LIN {X 0,Y 552.343,Z 361.925,A -85,B 0,C 180,E1 26679.853,E2 26679.853} C_VEL
LIN {X 0,Y 552.316,Z 361.93,A -85,B 0,C 180,E1 26676.515,E2 26676.515} C_VEL
LIN {X 0,Y 552.306,Z 361.936,A -85,B 0,C 180,E1 26673.143,E2 26673.143} C_VEL
LIN {X 0,Y 552.345,Z 361.928,A -85,B 0,C 180,E1 26669.855,E2 26669.855} C_VEL
LIN {X 0,Y 552.293,Z 361.931,A -85,B 0,C 180,E1 26666.589,E2 26666.589} C_VEL
LIN {X 0,Y 552.33,Z 361.932,A -85,B 0,C 180,E1 26663.244,E2 26663.244} C_VEL
LIN {X 0,Y 552.306,Z 361.932,A -85,B 0,C 180,E1 26660.008,E2 26660.008} C_VEL
LIN {X 0,Y 552.29,Z 361.935,A -85,B 0,C 180,E1 26656.621,E2 26656.621} C_VEL
LIN {X 0,Y 552.342,Z 361.931,A -85,B 0,C 180,E1 26653.398,E2 26653.398} C_VEL
LIN {X 0,Y 552.279,Z 361.932,A -85,B 0,C 180,E1 26650.22,E2 26650.22} C_VEL
LIN {X 0,Y 552.338,Z 361.933,A -85,B 0,C 180,E1 26646.967,E2 26646.967} C_VEL
LIN {X 0,Y 552.28,Z 361.935,A -85,B 0,C 180,E1 26643.737,E2 26643.737} C_VEL
LIN {X 0,Y 552.285,Z 361.937,A -85,B 0,C 180,E1 26640.311,E2 26640.311} C_VEL
LIN {X 0,Y 552.292,Z 361.933,A -85,B 0,C 180,E1 26637.302,E2 26637.302} C_VEL
LIN {X 0,Y 552.269,Z 361.935,A -85,B 0,C 180,E1 26633.973,E2 26633.973} C_VEL
LIN {X 0,Y 552.307,Z 361.936,A -85,B 0,C 180,E1 26630.939,E2 26630.939} C_VEL
LIN {X 0,Y 552.259,Z 361.937,A -85,B 0,C 180,E1 26627.665,E2 26627.665} C_VEL
LIN {X 0,Y 552.332,Z 361.933,A -85,B 0,C 180,E1 26624.46,E2 26624.46} C_VEL
LIN {X 0,Y 552.255,Z 361.936,A -85,B 0,C 180,E1 26621.227,E2 26621.227} C_VEL
LIN {X 0,Y 552.295,Z 361.933,A -85,B 0,C 180,E1 26617.945,E2 26617.945} C_VEL
LIN {X 0,Y 552.264,Z 361.927,A -85,B 0,C 180,E1 26614.935,E2 26614.935} C_VEL
LIN {X 0,Y 552.281,Z 361.934,A -85,B 0,C 180,E1 26611.567,E2 26611.567} C_VEL
LIN {X 0,Y 552.273,Z 361.928,A -85,B 0,C 180,E1 26608.695,E2 26608.695} C_VEL
LIN {X 0,Y 552.276,Z 361.929,A -85,B 0,C 180,E1 26605.23,E2 26605.23} C_VEL
LIN {X 0,Y 552.317,Z 361.938,A -85,B 0,C 180,E1 26602.112,E2 26602.112} C_VEL
LIN {X 0,Y 552.276,Z 361.935,A -85,B 0,C 180,E1 26598.857,E2 26598.857} C_VEL
LIN {X 0,Y 552.345,Z 361.921,A -85,B 0,C 180,E1 26595.64,E2 26595.64} C_VEL
LIN {X 0,Y 552.28,Z 361.923,A -85,B 0,C 180,E1 26592.384,E2 26592.384} C_VEL
LIN {X 0,Y 552.364,Z 362.227,A -85,B 0,C 180,E1 26591.86,E2 26591.86} C_VEL
LIN {X 0,Y 554.756,Z 368.091,A -85,B 0,C 180,E1 26591.269,E2 26591.269} C_VEL
LIN {X 0,Y 560.698,Z 379.842,A -85,B 0,C 180,E1 26590.068,E2 26590.068} C_VEL
LIN {X 0,Y 561.621,Z 381.954,A -85,B 0,C 180,E1 26589.855,E2 26589.855} C_VEL
LIN {X 0,Y 560.215,Z 433.691,A -85,B 0,C 180,E1 26586.78,E2 26586.78} C_VEL
LIN {X 0,Y 559.86,Z 455.296,A -85,B 0,C 180,E1 26585.548,E2 26585.548} C_VEL
LIN {X 0,Y 561.193,Z 465.51,A -85,B 0,C 180,E1 26585.289,E2 26585.289} C_VEL
LIN {X 0,Y 559.582,Z 691.156,A -85,B 0,C 180,E1 26581.995,E2 26581.995} C_VEL
LIN {X 0,Y 559.04,Z 762.319,A -85,B 0,C 180,E1 26580.945,E2 26580.945} C_VEL
LIN {X 0,Y 558.579,Z 783.876,A -85,B 0,C 180,E1 26580.433,E2 26580.433} C_VEL
LIN {X 0,Y 558.05,Z 805.556,A -85,B 0,C 180,E1 26579.723,E2 26579.723} C_VEL
LIN {X 0,Y 557.439,Z 826.444,A -85,B 0,C 180,E1 26578.846,E2 26578.846} C_VEL
LIN {X 0,Y 556.74,Z 845.795,A -85,B 0,C 180,E1 26577.833,E2 26577.833} C_VEL
LIN {X 0,Y 555.982,Z 866.365,A -85,B 0,C 180,E1 26576.542,E2 26576.542} C_VEL
LIN {X 0,Y 555.24,Z 885.138,A -85,B 0,C 180,E1 26575.147,E2 26575.147} C_VEL
LIN {X 0,Y 554.547,Z 902.924,A -85,B 0,C 180,E1 26573.593,E2 26573.593} C_VEL
LIN {X 0,Y 553.91,Z 919.52,A -85,B 0,C 180,E1 26571.904,E2 26571.904} C_VEL
LIN {X 0,Y 553.324,Z 935.884,A -85,B 0,C 180,E1 26569.968,E2 26569.968} C_VEL
LIN {X 0,Y 552.863,Z 950.053,A -85,B 0,C 180,E1 26568.013,E2 26568.013} C_VEL
LIN {X 0,Y 552.505,Z 962.742,A -85,B 0,C 180,E1 26565.965,E2 26565.965} C_VEL
LIN {X 0,Y 552.256,Z 973.338,A -85,B 0,C 180,E1 26563.932,E2 26563.932} C_VEL
LIN {X 0,Y 552.08,Z 983.072,A -85,B 0,C 180,E1 26561.702,E2 26561.702} C_VEL
LIN {X 0,Y 551.98,Z 990.592,A -85,B 0,C 180,E1 26559.592,E2 26559.592} C_VEL
LIN {X 0,Y 551.925,Z 996.4,A -85,B 0,C 180,E1 26557.494,E2 26557.494} C_VEL
LIN {X 0,Y 551.904,Z 1000.985,A -85,B 0,C 180,E1 26555.301,E2 26555.301} C_VEL
LIN {X 0,Y 551.907,Z 1003.785,A -85,B 0,C 180,E1 26553.22,E2 26553.22} C_VEL
LIN {X 0,Y 551.904,Z 1005.306,A -85,B 0,C 180,E1 26550.935,E2 26550.935} C_VEL
LIN {X 0,Y 551.909,Z 1005.238,A -85,B 0,C 180,E1 26548.755,E2 26548.755} C_VEL
LIN {X 0,Y 551.915,Z 1003.544,A -85,B 0,C 180,E1 26546.558,E2 26546.558} C_VEL
LIN {X 0,Y 551.924,Z 1000.222,A -85,B 0,C 180,E1 26544.283,E2 26544.283} C_VEL
LIN {X 0,Y 551.946,Z 995.639,A -85,B 0,C 180,E1 26542.193,E2 26542.193} C_VEL
LIN {X 0,Y 552.003,Z 989.18,A -85,B 0,C 180,E1 26539.987,E2 26539.987} C_VEL
LIN {X 0,Y 552.116,Z 981.437,A -85,B 0,C 180,E1 26537.875,E2 26537.875} C_VEL
LIN {X 0,Y 552.296,Z 971.783,A -85,B 0,C 180,E1 26535.748,E2 26535.748} C_VEL
LIN {X 0,Y 552.58,Z 960.206,A -85,B 0,C 180,E1 26533.606,E2 26533.606} C_VEL
LIN {X 0,Y 552.936,Z 947.891,A -85,B 0,C 180,E1 26531.663,E2 26531.663} C_VEL
LIN {X 0,Y 553.409,Z 933.339,A -85,B 0,C 180,E1 26529.705,E2 26529.705} C_VEL
LIN {X 0,Y 553.971,Z 917.685,A -85,B 0,C 180,E1 26527.897,E2 26527.897} C_VEL
LIN {X 0,Y 554.661,Z 899.915,A -85,B 0,C 180,E1 26526.131,E2 26526.131} C_VEL
LIN {X 0,Y 555.379,Z 881.773,A -85,B 0,C 180,E1 26524.588,E2 26524.588} C_VEL
LIN {X 0,Y 556.106,Z 863.135,A -85,B 0,C 180,E1 26523.235,E2 26523.235} C_VEL
LIN {X 0,Y 556.812,Z 843.818,A -85,B 0,C 180,E1 26522.055,E2 26522.055} C_VEL
LIN {X 0,Y 557.491,Z 823.944,A -85,B 0,C 180,E1 26521.041,E2 26521.041} C_VEL
LIN {X 0,Y 558.103,Z 804.103,A -85,B 0,C 180,E1 26520.222,E2 26520.222} C_VEL
LIN {X 0,Y 558.602,Z 782.228,A -85,B 0,C 180,E1 26519.521,E2 26519.521} C_VEL
LIN {X 0,Y 559.058,Z 760.348,A -85,B 0,C 180,E1 26519.022,E2 26519.022} C_VEL
LIN {X 0,Y 560.653,Z 537.271,A -85,B 0,C 180,E1 26515.768,E2 26515.768} C_VEL
LIN {X 0,Y 561.011,Z 462.845,A -85,B 0,C 180,E1 26514.657,E2 26514.657} C_VEL
LIN {X 0,Y 559.765,Z 453.839,A -85,B 0,C 180,E1 26514.392,E2 26514.392} C_VEL
LIN {X 0,Y 561.186,Z 397.807,A -85,B 0,C 180,E1 26511.099,E2 26511.099} C_VEL
LIN {X 0,Y 561.58,Z 381.583,A -85,B 0,C 180,E1 26510.118,E2 26510.118} C_VEL
LIN {X 0,Y 555.25,Z 369.007,A -85,B 0,C 180,E1 26508.825,E2 26508.825} C_VEL
LIN {X 0,Y 552.385,Z 362.34,A -85,B 0,C 180,E1 26508.161,E2 26508.161} C_VEL
LIN {X 0,Y 552.29,Z 361.923,A -85,B 0,C 180,E1 26507.811,E2 26507.811} C_VEL
LIN {X 0,Y 552.321,Z 361.927,A -85,B 0,C 180,E1 26504.654,E2 26504.654} C_VEL
LIN {X 0,Y 552.276,Z 361.935,A -85,B 0,C 180,E1 26501.361,E2 26501.361} C_VEL
LIN {X 0,Y 552.342,Z 361.936,A -85,B 0,C 180,E1 26498.118,E2 26498.118} C_VEL
LIN {X 0,Y 552.271,Z 361.93,A -85,B 0,C 180,E1 26494.897,E2 26494.897} C_VEL
LIN {X 0,Y 552.308,Z 361.928,A -85,B 0,C 180,E1 26491.668,E2 26491.668} C_VEL
LIN {X 0,Y 552.268,Z 361.934,A -85,B 0,C 180,E1 26488.67,E2 26488.67} C_VEL
LIN {X 0,Y 552.283,Z 361.926,A -85,B 0,C 180,E1 26485.293,E2 26485.293} C_VEL
LIN {X 0,Y 552.279,Z 361.932,A -85,B 0,C 180,E1 26482.233,E2 26482.233} C_VEL
LIN {X 0,Y 552.263,Z 361.936,A -85,B 0,C 180,E1 26478.909,E2 26478.909} C_VEL
LIN {X 0,Y 552.291,Z 361.939,A -85,B 0,C 180,E1 26475.864,E2 26475.864} C_VEL
LIN {X 0,Y 552.259,Z 361.938,A -85,B 0,C 180,E1 26472.644,E2 26472.644} C_VEL
LIN {X 0,Y 552.322,Z 361.937,A -85,B 0,C 180,E1 26469.482,E2 26469.482} C_VEL
LIN {X 0,Y 552.261,Z 361.935,A -85,B 0,C 180,E1 26466.34,E2 26466.34} C_VEL
LIN {X 0,Y 552.332,Z 361.932,A -85,B 0,C 180,E1 26463.113,E2 26463.113} C_VEL
LIN {X 0,Y 552.266,Z 361.937,A -85,B 0,C 180,E1 26460,E2 26460} C_VEL
LIN {X 0,Y 552.317,Z 361.935,A -85,B 0,C 180,E1 26456.723,E2 26456.723} C_VEL
LIN {X 0,Y 552.281,Z 361.931,A -85,B 0,C 180,E1 26453.555,E2 26453.555} C_VEL
LIN {X 0,Y 552.283,Z 361.931,A -85,B 0,C 180,E1 26450.096,E2 26450.096} C_VEL
LIN {X 0,Y 552.331,Z 361.938,A -85,B 0,C 180,E1 26446.922,E2 26446.922} C_VEL
LIN {X 0,Y 552.281,Z 361.935,A -85,B 0,C 180,E1 26443.703,E2 26443.703} C_VEL
LIN {X 0,Y 552.342,Z 361.933,A -85,B 0,C 180,E1 26440.434,E2 26440.434} C_VEL
LIN {X 0,Y 552.29,Z 361.934,A -85,B 0,C 180,E1 26437.206,E2 26437.206} C_VEL
LIN {X 0,Y 552.307,Z 361.93,A -85,B 0,C 180,E1 26433.786,E2 26433.786} C_VEL
LIN {X 0,Y 552.325,Z 361.933,A -85,B 0,C 180,E1 26432.641,E2 26432.641} C_VEL
LIN {X 0,Y 551.377,Z 362.054,A -85,B 0,C 180,E1 26431.841,E2 26431.841} C_VEL
LIN {X 0,Y 544.88,Z 362.854,A -85,B 0,C 180,E1 26429.597,E2 26429.597} C_VEL
LIN {X 0,Y 544.354,Z 362.92,A -85,B 0,C 180,E1 26429.012,E2 26429.012} C_VEL
LIN {X 0,Y 544.385,Z 362.919,A -85,B 0,C 180,E1 26425.677,E2 26425.677} C_VEL
LIN {X 0,Y 544.393,Z 362.912,A -85,B 0,C 180,E1 26422.327,E2 26422.327} C_VEL
LIN {X 0,Y 544.361,Z 362.922,A -85,B 0,C 180,E1 26419.01,E2 26419.01} C_VEL
LIN {X 0,Y 544.404,Z 362.907,A -85,B 0,C 180,E1 26415.74,E2 26415.74} C_VEL
LIN {X 0,Y 544.371,Z 362.925,A -85,B 0,C 180,E1 26412.408,E2 26412.408} C_VEL
LIN {X 0,Y 544.373,Z 362.924,A -85,B 0,C 180,E1 26408.909,E2 26408.909} C_VEL
LIN {X 0,Y 544.402,Z 362.924,A -85,B 0,C 180,E1 26405.548,E2 26405.548} C_VEL
LIN {X 0,Y 544.431,Z 363.119,A -85,B 0,C 180,E1 26403.177,E2 26403.177} C_VEL
LIN {X 0,Y 548.647,Z 375.762,A -85,B 0,C 180,E1 26401.572,E2 26401.572} C_VEL
LIN {X 0,Y 549.438,Z 378.934,A -85,B 0,C 180,E1 26401.237,E2 26401.237} C_VEL
LIN {X 0,Y 549.463,Z 383.628,A -85,B 0,C 180,E1 26400.87,E2 26400.87} C_VEL
LIN {X 0,Y 551.825,Z 395.845,A -85,B 0,C 180,E1 26400.533,E2 26400.533} C_VEL
LIN {X 0,Y 550.089,Z 643.165,A -85,B 0,C 180,E1 26397,E2 26397} C_VEL
LIN {X 0,Y 549.682,Z 663.581,A -85,B 0,C 180,E1 26396.524,E2 26396.524} C_VEL
LIN {X 0,Y 549.19,Z 683.218,A -85,B 0,C 180,E1 26395.877,E2 26395.877} C_VEL
LIN {X 0,Y 548.592,Z 703.287,A -85,B 0,C 180,E1 26395.011,E2 26395.011} C_VEL
LIN {X 0,Y 547.936,Z 721.879,A -85,B 0,C 180,E1 26394.009,E2 26394.009} C_VEL
LIN {X 0,Y 547.252,Z 740.465,A -85,B 0,C 180,E1 26392.786,E2 26392.786} C_VEL
LIN {X 0,Y 546.545,Z 758.589,A -85,B 0,C 180,E1 26391.347,E2 26391.347} C_VEL
LIN {X 0,Y 545.911,Z 774.895,A -85,B 0,C 180,E1 26389.803,E2 26389.803} C_VEL
LIN {X 0,Y 545.352,Z 789.659,A -85,B 0,C 180,E1 26388.158,E2 26388.158} C_VEL
LIN {X 0,Y 544.9,Z 803.014,A -85,B 0,C 180,E1 26386.412,E2 26386.412} C_VEL
LIN {X 0,Y 544.518,Z 815.631,A -85,B 0,C 180,E1 26384.459,E2 26384.459} C_VEL
LIN {X 0,Y 544.256,Z 826.628,A -85,B 0,C 180,E1 26382.41,E2 26382.41} C_VEL
LIN {X 0,Y 544.081,Z 835.589,A -85,B 0,C 180,E1 26380.374,E2 26380.374} C_VEL
LIN {X 0,Y 543.986,Z 843.067,A -85,B 0,C 180,E1 26378.241,E2 26378.241} C_VEL
LIN {X 0,Y 543.936,Z 848.903,A -85,B 0,C 180,E1 26376.013,E2 26376.013} C_VEL
LIN {X 0,Y 543.918,Z 852.677,A -85,B 0,C 180,E1 26373.899,E2 26373.899} C_VEL
LIN {X 0,Y 543.91,Z 854.847,A -85,B 0,C 180,E1 26371.79,E2 26371.79} C_VEL
LIN {X 0,Y 543.904,Z 855.449,A -85,B 0,C 180,E1 26369.684,E2 26369.684} C_VEL
LIN {X 0,Y 543.905,Z 854.492,A -85,B 0,C 180,E1 26367.577,E2 26367.577} C_VEL
LIN {X 0,Y 543.918,Z 851.699,A -85,B 0,C 180,E1 26365.361,E2 26365.361} C_VEL
LIN {X 0,Y 543.945,Z 847.346,A -85,B 0,C 180,E1 26363.244,E2 26363.244} C_VEL
LIN {X 0,Y 543.998,Z 841.271,A -85,B 0,C 180,E1 26361.119,E2 26361.119} C_VEL
LIN {X 0,Y 544.105,Z 833.793,A -85,B 0,C 180,E1 26359.09,E2 26359.09} C_VEL
LIN {X 0,Y 544.307,Z 824.452,A -85,B 0,C 180,E1 26357.051,E2 26357.051} C_VEL
LIN {X 0,Y 544.578,Z 813.591,A -85,B 0,C 180,E1 26355.106,E2 26355.106} C_VEL
LIN {X 0,Y 544.949,Z 801.32,A -85,B 0,C 180,E1 26353.26,E2 26353.26} C_VEL
LIN {X 0,Y 545.419,Z 787.628,A -85,B 0,C 180,E1 26351.511,E2 26351.511} C_VEL
LIN {X 0,Y 546.016,Z 771.787,A -85,B 0,C 180,E1 26349.796,E2 26349.796} C_VEL
LIN {X 0,Y 546.675,Z 755.081,A -85,B 0,C 180,E1 26348.269,E2 26348.269} C_VEL
LIN {X 0,Y 547.359,Z 737.607,A -85,B 0,C 180,E1 26346.925,E2 26346.925} C_VEL
LIN {X 0,Y 548.021,Z 719.612,A -85,B 0,C 180,E1 26345.765,E2 26345.765} C_VEL
LIN {X 0,Y 548.681,Z 700.505,A -85,B 0,C 180,E1 26344.762,E2 26344.762} C_VEL
LIN {X 0,Y 549.259,Z 681.058,A -85,B 0,C 180,E1 26343.952,E2 26343.952} C_VEL
LIN {X 0,Y 549.733,Z 660.673,A -85,B 0,C 180,E1 26343.307,E2 26343.307} C_VEL
LIN {X 0,Y 550.118,Z 639.409,A -85,B 0,C 180,E1 26342.848,E2 26342.848} C_VEL
LIN {X 0,Y 551.822,Z 394.728,A -85,B 0,C 180,E1 26339.361,E2 26339.361} C_VEL
LIN {X 0,Y 549.369,Z 382.831,A -85,B 0,C 180,E1 26339.001,E2 26339.001} C_VEL
LIN {X 0,Y 549.407,Z 378.116,A -85,B 0,C 180,E1 26338.598,E2 26338.598} C_VEL
LIN {X 0,Y 544.904,Z 364.895,A -85,B 0,C 180,E1 26336.989,E2 26336.989} C_VEL
LIN {X 0,Y 544.412,Z 363.01,A -85,B 0,C 180,E1 26336.695,E2 26336.695} C_VEL
LIN {X 0,Y 544.373,Z 362.914,A -85,B 0,C 180,E1 26333.353,E2 26333.353} C_VEL
LIN {X 0,Y 544.403,Z 362.917,A -85,B 0,C 180,E1 26329.985,E2 26329.985} C_VEL
LIN {X 0,Y 544.403,Z 362.92,A -85,B 0,C 180,E1 26326.508,E2 26326.508} C_VEL
LIN {X 0,Y 544.366,Z 362.921,A -85,B 0,C 180,E1 26323.187,E2 26323.187} C_VEL
LIN {X 0,Y 544.404,Z 362.912,A -85,B 0,C 180,E1 26319.858,E2 26319.858} C_VEL
LIN {X 0,Y 544.376,Z 362.919,A -85,B 0,C 180,E1 26316.519,E2 26316.519} C_VEL
LIN {X 0,Y 544.363,Z 362.925,A -85,B 0,C 180,E1 26313.06,E2 26313.06} C_VEL
LIN {X 0,Y 544.406,Z 362.918,A -85,B 0,C 180,E1 26309.728,E2 26309.728} C_VEL
LIN {X 0,Y 544.356,Z 362.92,A -85,B 0,C 180,E1 26306.509,E2 26306.509} C_VEL
LIN {X 0,Y 544.381,Z 362.922,A -85,B 0,C 180,E1 26303.145,E2 26303.145} C_VEL
LIN {X 0,Y 544.379,Z 362.92,A -85,B 0,C 180,E1 26299.864,E2 26299.864} C_VEL
LIN {X 0,Y 544.348,Z 362.924,A -85,B 0,C 180,E1 26296.52,E2 26296.52} C_VEL
LIN {X 0,Y 544.407,Z 362.921,A -85,B 0,C 180,E1 26293.268,E2 26293.268} C_VEL
LIN {X 0,Y 544.342,Z 362.92,A -85,B 0,C 180,E1 26290.05,E2 26290.05} C_VEL
LIN {X 0,Y 544.375,Z 362.92,A -85,B 0,C 180,E1 26286.751,E2 26286.751} C_VEL
LIN {X 0,Y 544.35,Z 362.924,A -85,B 0,C 180,E1 26283.581,E2 26283.581} C_VEL
LIN {X 0,Y 544.338,Z 362.926,A -85,B 0,C 180,E1 26280.211,E2 26280.211} C_VEL
LIN {X 0,Y 544.379,Z 362.921,A -85,B 0,C 180,E1 26277.052,E2 26277.052} C_VEL
LIN {X 0,Y 544.325,Z 362.924,A -85,B 0,C 180,E1 26273.779,E2 26273.779} C_VEL
LIN {X 0,Y 544.394,Z 362.926,A -85,B 0,C 180,E1 26270.592,E2 26270.592} C_VEL
LIN {X 0,Y 544.322,Z 362.926,A -85,B 0,C 180,E1 26267.374,E2 26267.374} C_VEL
LIN {X 0,Y 544.344,Z 362.928,A -85,B 0,C 180,E1 26264.007,E2 26264.007} C_VEL
LIN {X 0,Y 544.333,Z 362.924,A -85,B 0,C 180,E1 26260.916,E2 26260.916} C_VEL
LIN {X 0,Y 544.323,Z 362.921,A -85,B 0,C 180,E1 26257.498,E2 26257.498} C_VEL
LIN {X 0,Y 544.385,Z 362.915,A -85,B 0,C 180,E1 26254.313,E2 26254.313} C_VEL
LIN {X 0,Y 544.324,Z 362.924,A -85,B 0,C 180,E1 26251.112,E2 26251.112} C_VEL
LIN {X 0,Y 544.399,Z 362.92,A -85,B 0,C 180,E1 26247.942,E2 26247.942} C_VEL
LIN {X 0,Y 544.332,Z 362.918,A -85,B 0,C 180,E1 26244.776,E2 26244.776} C_VEL
LIN {X 0,Y 544.372,Z 362.922,A -85,B 0,C 180,E1 26241.478,E2 26241.478} C_VEL
LIN {X 0,Y 544.351,Z 362.925,A -85,B 0,C 180,E1 26238.324,E2 26238.324} C_VEL
LIN {X 0,Y 544.351,Z 362.922,A -85,B 0,C 180,E1 26234.996,E2 26234.996} C_VEL
LIN {X 0,Y 544.375,Z 363.16,A -85,B 0,C 180,E1 26232.45,E2 26232.45} C_VEL
LIN {X 0,Y 545.681,Z 366.42,A -85,B 0,C 180,E1 26232.091,E2 26232.091} C_VEL
LIN {X 0,Y 555.056,Z 385.798,A -85,B 0,C 180,E1 26230.175,E2 26230.175} C_VEL
LIN {X 0,Y 553.444,Z 437.914,A -85,B 0,C 180,E1 26227.046,E2 26227.046} C_VEL
LIN {X 0,Y 553.129,Z 455.298,A -85,B 0,C 180,E1 26226.048,E2 26226.048} C_VEL
LIN {X 0,Y 554.65,Z 466.908,A -85,B 0,C 180,E1 26225.747,E2 26225.747} C_VEL
LIN {X 0,Y 552.786,Z 692.683,A -85,B 0,C 180,E1 26222.413,E2 26222.413} C_VEL
LIN {X 0,Y 552.171,Z 762.512,A -85,B 0,C 180,E1 26221.369,E2 26221.369} C_VEL
LIN {X 0,Y 551.64,Z 784.137,A -85,B 0,C 180,E1 26220.849,E2 26220.849} C_VEL
LIN {X 0,Y 551.017,Z 806.292,A -85,B 0,C 180,E1 26220.111,E2 26220.111} C_VEL
LIN {X 0,Y 550.331,Z 826.443,A -85,B 0,C 180,E1 26219.254,E2 26219.254} C_VEL
LIN {X 0,Y 549.538,Z 845.798,A -85,B 0,C 180,E1 26218.23,E2 26218.23} C_VEL
LIN {X 0,Y 548.656,Z 866.361,A -85,B 0,C 180,E1 26216.925,E2 26216.925} C_VEL
LIN {X 0,Y 547.804,Z 885.135,A -85,B 0,C 180,E1 26215.513,E2 26215.513} C_VEL
LIN {X 0,Y 547.003,Z 902.926,A -85,B 0,C 180,E1 26213.939,E2 26213.939} C_VEL
LIN {X 0,Y 546.265,Z 919.196,A -85,B 0,C 180,E1 26212.263,E2 26212.263} C_VEL
LIN {X 0,Y 545.603,Z 935.035,A -85,B 0,C 180,E1 26210.375,E2 26210.375} C_VEL
LIN {X 0,Y 545.096,Z 948.639,A -85,B 0,C 180,E1 26208.5,E2 26208.5} C_VEL
LIN {X 0,Y 544.662,Z 961.471,A -85,B 0,C 180,E1 26206.42,E2 26206.42} C_VEL
LIN {X 0,Y 544.34,Z 972.82,A -85,B 0,C 180,E1 26204.248,E2 26204.248} C_VEL
LIN {X 0,Y 544.135,Z 982.257,A -85,B 0,C 180,E1 26202.091,E2 26202.091} C_VEL
LIN {X 0,Y 544.009,Z 989.886,A -85,B 0,C 180,E1 26199.948,E2 26199.948} C_VEL
LIN {X 0,Y 543.942,Z 996.146,A -85,B 0,C 180,E1 26197.711,E2 26197.711} C_VEL
LIN {X 0,Y 543.915,Z 1000.824,A -85,B 0,C 180,E1 26195.485,E2 26195.485} C_VEL
LIN {X 0,Y 543.91,Z 1003.785,A -85,B 0,C 180,E1 26193.267,E2 26193.267} C_VEL
LIN {X 0,Y 543.905,Z 1005.306,A -85,B 0,C 180,E1 26190.948,E2 26190.948} C_VEL
LIN {X 0,Y 543.908,Z 1005.238,A -85,B 0,C 180,E1 26188.736,E2 26188.736} C_VEL
LIN {X 0,Y 543.913,Z 1003.56,A -85,B 0,C 180,E1 26186.523,E2 26186.523} C_VEL
LIN {X 0,Y 543.927,Z 1000.222,A -85,B 0,C 180,E1 26184.198,E2 26184.198} C_VEL
LIN {X 0,Y 543.958,Z 995.639,A -85,B 0,C 180,E1 26182.077,E2 26182.077} C_VEL
LIN {X 0,Y 544.03,Z 989.181,A -85,B 0,C 180,E1 26179.839,E2 26179.839} C_VEL
LIN {X 0,Y 544.161,Z 981.436,A -85,B 0,C 180,E1 26177.695,E2 26177.695} C_VEL
LIN {X 0,Y 544.377,Z 971.784,A -85,B 0,C 180,E1 26175.537,E2 26175.537} C_VEL
LIN {X 0,Y 544.706,Z 960.206,A -85,B 0,C 180,E1 26173.362,E2 26173.362} C_VEL
LIN {X 0,Y 545.123,Z 947.889,A -85,B 0,C 180,E1 26171.391,E2 26171.391} C_VEL
LIN {X 0,Y 545.673,Z 933.34,A -85,B 0,C 180,E1 26169.405,E2 26169.405} C_VEL
LIN {X 0,Y 546.304,Z 918.191,A -85,B 0,C 180,E1 26167.627,E2 26167.627} C_VEL
LIN {X 0,Y 547.107,Z 900.519,A -85,B 0,C 180,E1 26165.838,E2 26165.838} C_VEL
LIN {X 0,Y 547.914,Z 883.071,A -85,B 0,C 180,E1 26164.32,E2 26164.32} C_VEL
LIN {X 0,Y 548.728,Z 864.64,A -85,B 0,C 180,E1 26162.954,E2 26162.954} C_VEL
LIN {X 0,Y 549.583,Z 844.709,A -85,B 0,C 180,E1 26161.707,E2 26161.707} C_VEL
LIN {X 0,Y 550.38,Z 824.652,A -85,B 0,C 180,E1 26160.663,E2 26160.663} C_VEL
LIN {X 0,Y 551.074,Z 804.84,A -85,B 0,C 180,E1 26159.833,E2 26159.833} C_VEL
LIN {X 0,Y 551.669,Z 782.618,A -85,B 0,C 180,E1 26159.108,E2 26159.108} C_VEL
LIN {X 0,Y 552.189,Z 760.883,A -85,B 0,C 180,E1 26158.602,E2 26158.602} C_VEL
LIN {X 0,Y 554.023,Z 539.306,A -85,B 0,C 180,E1 26155.332,E2 26155.332} C_VEL
LIN {X 0,Y 554.48,Z 464.261,A -85,B 0,C 180,E1 26154.199,E2 26154.199} C_VEL
LIN {X 0,Y 553.035,Z 453.865,A -85,B 0,C 180,E1 26153.891,E2 26153.891} C_VEL
LIN {X 0,Y 554.652,Z 398.862,A -85,B 0,C 180,E1 26150.619,E2 26150.619} C_VEL
LIN {X 0,Y 555.03,Z 385.441,A -85,B 0,C 180,E1 26149.801,E2 26149.801} C_VEL
LIN {X 0,Y 546.189,Z 367.32,A -85,B 0,C 180,E1 26148.007,E2 26148.007} C_VEL
LIN {X 0,Y 544.414,Z 363.375,A -85,B 0,C 180,E1 26147.587,E2 26147.587} C_VEL
LIN {X 0,Y 544.341,Z 362.909,A -85,B 0,C 180,E1 26147.284,E2 26147.284} C_VEL
LIN {X 0,Y 544.37,Z 362.912,A -85,B 0,C 180,E1 26143.952,E2 26143.952} C_VEL
LIN {X 0,Y 544.351,Z 362.919,A -85,B 0,C 180,E1 26140.828,E2 26140.828} C_VEL
LIN {X 0,Y 544.341,Z 362.926,A -85,B 0,C 180,E1 26137.444,E2 26137.444} C_VEL
LIN {X 0,Y 544.391,Z 362.917,A -85,B 0,C 180,E1 26134.195,E2 26134.195} C_VEL
LIN {X 0,Y 544.326,Z 362.915,A -85,B 0,C 180,E1 26130.938,E2 26130.938} C_VEL
LIN {X 0,Y 544.383,Z 362.928,A -85,B 0,C 180,E1 26127.689,E2 26127.689} C_VEL
LIN {X 0,Y 544.325,Z 362.913,A -85,B 0,C 180,E1 26124.528,E2 26124.528} C_VEL
LIN {X 0,Y 544.334,Z 362.928,A -85,B 0,C 180,E1 26121.09,E2 26121.09} C_VEL
LIN {X 0,Y 544.35,Z 362.924,A -85,B 0,C 180,E1 26117.973,E2 26117.973} C_VEL
LIN {X 0,Y 544.317,Z 362.926,A -85,B 0,C 180,E1 26114.684,E2 26114.684} C_VEL
LIN {X 0,Y 544.389,Z 362.921,A -85,B 0,C 180,E1 26111.441,E2 26111.441} C_VEL
LIN {X 0,Y 544.319,Z 362.926,A -85,B 0,C 180,E1 26108.237,E2 26108.237} C_VEL
LIN {X 0,Y 544.383,Z 362.925,A -85,B 0,C 180,E1 26105.058,E2 26105.058} C_VEL
LIN {X 0,Y 544.331,Z 362.923,A -85,B 0,C 180,E1 26101.894,E2 26101.894} C_VEL
LIN {X 0,Y 544.35,Z 362.919,A -85,B 0,C 180,E1 26098.526,E2 26098.526} C_VEL
LIN {X 0,Y 544.36,Z 362.926,A -85,B 0,C 180,E1 26095.364,E2 26095.364} C_VEL
LIN {X 0,Y 544.339,Z 362.924,A -85,B 0,C 180,E1 26092.081,E2 26092.081} C_VEL
LIN {X 0,Y 544.398,Z 362.92,A -85,B 0,C 180,E1 26088.881,E2 26088.881} C_VEL
LIN {X 0,Y 544.338,Z 362.922,A -85,B 0,C 180,E1 26085.642,E2 26085.642} C_VEL
LIN {X 0,Y 544.395,Z 362.92,A -85,B 0,C 180,E1 26082.359,E2 26082.359} C_VEL
LIN {X 0,Y 544.355,Z 362.925,A -85,B 0,C 180,E1 26079.125,E2 26079.125} C_VEL
LIN {X 0,Y 544.352,Z 362.922,A -85,B 0,C 180,E1 26075.637,E2 26075.637} C_VEL
LIN {X 0,Y 544.405,Z 362.921,A -85,B 0,C 180,E1 26072.43,E2 26072.43} C_VEL
LIN {X 0,Y 544.353,Z 362.919,A -85,B 0,C 180,E1 26069.172,E2 26069.172} C_VEL
LIN {X 0,Y 544.354,Z 362.92,A -85,B 0,C 180,E1 26069.012,E2 26069.012} C_VEL
LIN {X 0,Y 543.393,Z 363.05,A -85,B 0,C 180,E1 26068.202,E2 26068.202} C_VEL
LIN {X 0,Y 536.877,Z 363.856,A -85,B 0,C 180,E1 26065.865,E2 26065.865} C_VEL
LIN {X 0,Y 536.422,Z 363.91,A -85,B 0,C 180,E1 26065.331,E2 26065.331} C_VEL
LIN {X 0,Y 536.465,Z 363.892,A -85,B 0,C 180,E1 26062.027,E2 26062.027} C_VEL
LIN {X 0,Y 536.426,Z 363.913,A -85,B 0,C 180,E1 26058.684,E2 26058.684} C_VEL
LIN {X 0,Y 536.437,Z 363.9,A -85,B 0,C 180,E1 26055.207,E2 26055.207} C_VEL
LIN {X 0,Y 536.462,Z 363.897,A -85,B 0,C 180,E1 26051.849,E2 26051.849} C_VEL
LIN {X 0,Y 536.429,Z 363.915,A -85,B 0,C 180,E1 26048.478,E2 26048.478} C_VEL
LIN {X 0,Y 536.453,Z 363.909,A -85,B 0,C 180,E1 26045.029,E2 26045.029} C_VEL
LIN {X 0,Y 536.497,Z 364.158,A -85,B 0,C 180,E1 26043.732,E2 26043.732} C_VEL
LIN {X 0,Y 541.522,Z 378.665,A -85,B 0,C 180,E1 26041.86,E2 26041.86} C_VEL
LIN {X 0,Y 542.341,Z 381.653,A -85,B 0,C 180,E1 26041.507,E2 26041.507} C_VEL
LIN {X 0,Y 542.494,Z 384.417,A -85,B 0,C 180,E1 26041.32,E2 26041.32} C_VEL
LIN {X 0,Y 544.927,Z 397.237,A -85,B 0,C 180,E1 26040.941,E2 26040.941} C_VEL
LIN {X 0,Y 542.962,Z 642.994,A -85,B 0,C 180,E1 26037.387,E2 26037.387} C_VEL
LIN {X 0,Y 542.502,Z 663.463,A -85,B 0,C 180,E1 26036.907,E2 26036.907} C_VEL
LIN {X 0,Y 541.952,Z 683.236,A -85,B 0,C 180,E1 26036.249,E2 26036.249} C_VEL
LIN {X 0,Y 541.268,Z 703.299,A -85,B 0,C 180,E1 26035.373,E2 26035.373} C_VEL
LIN {X 0,Y 540.524,Z 721.888,A -85,B 0,C 180,E1 26034.359,E2 26034.359} C_VEL
LIN {X 0,Y 539.754,Z 740.473,A -85,B 0,C 180,E1 26033.121,E2 26033.121} C_VEL
LIN {X 0,Y 538.948,Z 758.6,A -85,B 0,C 180,E1 26031.663,E2 26031.663} C_VEL
LIN {X 0,Y 538.22,Z 774.903,A -85,B 0,C 180,E1 26030.099,E2 26030.099} C_VEL
LIN {X 0,Y 537.577,Z 789.664,A -85,B 0,C 180,E1 26028.43,E2 26028.43} C_VEL
LIN {X 0,Y 537.057,Z 803.018,A -85,B 0,C 180,E1 26026.659,E2 26026.659} C_VEL
LIN {X 0,Y 536.617,Z 815.633,A -85,B 0,C 180,E1 26024.677,E2 26024.677} C_VEL
LIN {X 0,Y 536.313,Z 826.632,A -85,B 0,C 180,E1 26022.597,E2 26022.597} C_VEL
LIN {X 0,Y 536.113,Z 835.593,A -85,B 0,C 180,E1 26020.53,E2 26020.53} C_VEL
LIN {X 0,Y 536,Z 843.069,A -85,B 0,C 180,E1 26018.365,E2 26018.365} C_VEL
LIN {X 0,Y 535.94,Z 848.905,A -85,B 0,C 180,E1 26016.103,E2 26016.103} C_VEL
LIN {X 0,Y 535.919,Z 852.678,A -85,B 0,C 180,E1 26013.958,E2 26013.958} C_VEL
LIN {X 0,Y 535.911,Z 854.847,A -85,B 0,C 180,E1 26011.817,E2 26011.817} C_VEL
LIN {X 0,Y 535.904,Z 855.449,A -85,B 0,C 180,E1 26009.679,E2 26009.679} C_VEL
LIN {X 0,Y 535.905,Z 854.491,A -85,B 0,C 180,E1 26007.54,E2 26007.54} C_VEL
LIN {X 0,Y 535.919,Z 851.857,A -85,B 0,C 180,E1 26005.399,E2 26005.399} C_VEL
LIN {X 0,Y 535.948,Z 847.599,A -85,B 0,C 180,E1 26003.251,E2 26003.251} C_VEL
LIN {X 0,Y 536.009,Z 841.623,A -85,B 0,C 180,E1 26001.094,E2 26001.094} C_VEL
LIN {X 0,Y 536.132,Z 834.248,A -85,B 0,C 180,E1 25999.035,E2 25999.035} C_VEL
LIN {X 0,Y 536.356,Z 824.977,A -85,B 0,C 180,E1 25996.965,E2 25996.965} C_VEL
LIN {X 0,Y 536.665,Z 814.228,A -85,B 0,C 180,E1 25994.992,E2 25994.992} C_VEL
LIN {X 0,Y 537.087,Z 802.055,A -85,B 0,C 180,E1 25993.114,E2 25993.114} C_VEL
LIN {X 0,Y 537.619,Z 788.549,A -85,B 0,C 180,E1 25991.346,E2 25991.346} C_VEL
LIN {X 0,Y 538.269,Z 773.57,A -85,B 0,C 180,E1 25989.676,E2 25989.676} C_VEL
LIN {X 0,Y 538.986,Z 757.656,A -85,B 0,C 180,E1 25988.166,E2 25988.166} C_VEL
LIN {X 0,Y 539.782,Z 739.877,A -85,B 0,C 180,E1 25986.746,E2 25986.746} C_VEL
LIN {X 0,Y 540.552,Z 721.268,A -85,B 0,C 180,E1 25985.513,E2 25985.513} C_VEL
LIN {X 0,Y 541.283,Z 702.754,A -85,B 0,C 180,E1 25984.51,E2 25984.51} C_VEL
LIN {X 0,Y 541.933,Z 683.811,A -85,B 0,C 180,E1 25983.683,E2 25983.683} C_VEL
LIN {X 0,Y 542.499,Z 663.774,A -85,B 0,C 180,E1 25983.011,E2 25983.011} C_VEL
LIN {X 0,Y 542.961,Z 643.267,A -85,B 0,C 180,E1 25982.527,E2 25982.527} C_VEL
LIN {X 0,Y 544.914,Z 398.88,A -85,B 0,C 180,E1 25978.993,E2 25978.993} C_VEL
LIN {X 0,Y 544.609,Z 394.681,A -85,B 0,C 180,E1 25978.909,E2 25978.909} C_VEL
LIN {X 0,Y 542.322,Z 383.07,A -85,B 0,C 180,E1 25978.522,E2 25978.522} C_VEL
LIN {X 0,Y 542.049,Z 380.311,A -85,B 0,C 180,E1 25978.251,E2 25978.251} C_VEL
LIN {X 0,Y 537.617,Z 367.183,A -85,B 0,C 180,E1 25976.602,E2 25976.602} C_VEL
LIN {X 0,Y 536.482,Z 364.044,A -85,B 0,C 180,E1 25976.137,E2 25976.137} C_VEL
LIN {X 0,Y 536.459,Z 363.894,A -85,B 0,C 180,E1 25972.722,E2 25972.722} C_VEL
LIN {X 0,Y 536.43,Z 363.899,A -85,B 0,C 180,E1 25969.342,E2 25969.342} C_VEL
LIN {X 0,Y 536.462,Z 363.911,A -85,B 0,C 180,E1 25965.962,E2 25965.962} C_VEL
LIN {X 0,Y 536.45,Z 363.906,A -85,B 0,C 180,E1 25962.577,E2 25962.577} C_VEL
LIN {X 0,Y 536.424,Z 363.893,A -85,B 0,C 180,E1 25959.166,E2 25959.166} C_VEL
LIN {X 0,Y 536.466,Z 363.912,A -85,B 0,C 180,E1 25955.819,E2 25955.819} C_VEL
LIN {X 0,Y 536.431,Z 363.911,A -85,B 0,C 180,E1 25952.467,E2 25952.467} C_VEL
LIN {X 0,Y 536.424,Z 363.914,A -85,B 0,C 180,E1 25948.988,E2 25948.988} C_VEL
LIN {X 0,Y 536.464,Z 363.907,A -85,B 0,C 180,E1 25945.739,E2 25945.739} C_VEL
LIN {X 0,Y 536.412,Z 363.909,A -85,B 0,C 180,E1 25942.415,E2 25942.415} C_VEL
LIN {X 0,Y 536.439,Z 363.91,A -85,B 0,C 180,E1 25939.037,E2 25939.037} C_VEL
LIN {X 0,Y 536.434,Z 363.91,A -85,B 0,C 180,E1 25935.791,E2 25935.791} C_VEL
LIN {X 0,Y 536.406,Z 363.914,A -85,B 0,C 180,E1 25932.408,E2 25932.408} C_VEL
LIN {X 0,Y 536.465,Z 363.91,A -85,B 0,C 180,E1 25929.116,E2 25929.116} C_VEL
LIN {X 0,Y 536.4,Z 363.907,A -85,B 0,C 180,E1 25925.885,E2 25925.885} C_VEL
LIN {X 0,Y 536.415,Z 363.909,A -85,B 0,C 180,E1 25922.457,E2 25922.457} C_VEL
LIN {X 0,Y 536.416,Z 363.914,A -85,B 0,C 180,E1 25919.359,E2 25919.359} C_VEL
LIN {X 0,Y 536.394,Z 363.915,A -85,B 0,C 180,E1 25916.045,E2 25916.045} C_VEL
LIN {X 0,Y 536.451,Z 363.909,A -85,B 0,C 180,E1 25912.827,E2 25912.827} C_VEL
LIN {X 0,Y 536.382,Z 363.914,A -85,B 0,C 180,E1 25909.583,E2 25909.583} C_VEL
LIN {X 0,Y 536.432,Z 363.914,A -85,B 0,C 180,E1 25906.307,E2 25906.307} C_VEL
LIN {X 0,Y 536.38,Z 363.917,A -85,B 0,C 180,E1 25903.206,E2 25903.206} C_VEL
LIN {X 0,Y 536.399,Z 363.917,A -85,B 0,C 180,E1 25899.828,E2 25899.828} C_VEL
LIN {X 0,Y 536.4,Z 363.907,A -85,B 0,C 180,E1 25896.762,E2 25896.762} C_VEL
LIN {X 0,Y 536.39,Z 363.917,A -85,B 0,C 180,E1 25893.425,E2 25893.425} C_VEL
LIN {X 0,Y 536.439,Z 363.9,A -85,B 0,C 180,E1 25890.278,E2 25890.278} C_VEL
LIN {X 0,Y 536.39,Z 363.917,A -85,B 0,C 180,E1 25887.008,E2 25887.008} C_VEL
LIN {X 0,Y 536.452,Z 363.899,A -85,B 0,C 180,E1 25883.784,E2 25883.784} C_VEL
LIN {X 0,Y 536.396,Z 363.912,A -85,B 0,C 180,E1 25880.669,E2 25880.669} C_VEL
LIN {X 0,Y 536.44,Z 363.911,A -85,B 0,C 180,E1 25877.406,E2 25877.406} C_VEL
LIN {X 0,Y 536.417,Z 363.92,A -85,B 0,C 180,E1 25874.191,E2 25874.191} C_VEL
LIN {X 0,Y 536.449,Z 364.118,A -85,B 0,C 180,E1 25873.061,E2 25873.061} C_VEL
LIN {X 0,Y 537.174,Z 366.462,A -85,B 0,C 180,E1 25872.791,E2 25872.791} C_VEL
LIN {X 0,Y 548.249,Z 389.216,A -85,B 0,C 180,E1 25870.48,E2 25870.48} C_VEL
LIN {X 0,Y 547.221,Z 426.299,A -85,B 0,C 180,E1 25868.269,E2 25868.269} C_VEL
LIN {X 0,Y 546.421,Z 455.21,A -85,B 0,C 180,E1 25866.565,E2 25866.565} C_VEL
LIN {X 0,Y 548.144,Z 468.258,A -85,B 0,C 180,E1 25866.216,E2 25866.216} C_VEL
LIN {X 0,Y 546.023,Z 693.955,A -85,B 0,C 180,E1 25862.846,E2 25862.846} C_VEL
LIN {X 0,Y 545.336,Z 762.512,A -85,B 0,C 180,E1 25861.808,E2 25861.808} C_VEL
LIN {X 0,Y 544.738,Z 784.137,A -85,B 0,C 180,E1 25861.284,E2 25861.284} C_VEL
LIN {X 0,Y 544.041,Z 806.289,A -85,B 0,C 180,E1 25860.538,E2 25860.538} C_VEL
LIN {X 0,Y 543.253,Z 826.442,A -85,B 0,C 180,E1 25859.673,E2 25859.673} C_VEL
LIN {X 0,Y 542.364,Z 845.801,A -85,B 0,C 180,E1 25858.638,E2 25858.638} C_VEL
LIN {X 0,Y 541.362,Z 866.175,A -85,B 0,C 180,E1 25857.331,E2 25857.331} C_VEL
LIN {X 0,Y 540.403,Z 885.133,A -85,B 0,C 180,E1 25855.888,E2 25855.888} C_VEL
LIN {X 0,Y 539.48,Z 902.927,A -85,B 0,C 180,E1 25854.294,E2 25854.294} C_VEL
LIN {X 0,Y 538.628,Z 919.196,A -85,B 0,C 180,E1 25852.596,E2 25852.596} C_VEL
LIN {X 0,Y 537.868,Z 935.035,A -85,B 0,C 180,E1 25850.681,E2 25850.681} C_VEL
LIN {X 0,Y 537.262,Z 949.194,A -85,B 0,C 180,E1 25848.692,E2 25848.692} C_VEL
LIN {X 0,Y 536.792,Z 961.469,A -85,B 0,C 180,E1 25846.668,E2 25846.668} C_VEL
LIN {X 0,Y 536.42,Z 972.821,A -85,B 0,C 180,E1 25844.463,E2 25844.463} C_VEL
LIN {X 0,Y 536.18,Z 982.258,A -85,B 0,C 180,E1 25842.273,E2 25842.273} C_VEL
LIN {X 0,Y 536.036,Z 989.885,A -85,B 0,C 180,E1 25840.098,E2 25840.098} C_VEL
LIN {X 0,Y 535.956,Z 996.146,A -85,B 0,C 180,E1 25837.827,E2 25837.827} C_VEL
LIN {X 0,Y 535.921,Z 1000.824,A -85,B 0,C 180,E1 25835.567,E2 25835.567} C_VEL
LIN {X 0,Y 535.911,Z 1003.786,A -85,B 0,C 180,E1 25833.316,E2 25833.316} C_VEL
LIN {X 0,Y 535.905,Z 1005.306,A -85,B 0,C 180,E1 25830.962,E2 25830.962} C_VEL
LIN {X 0,Y 535.907,Z 1005.237,A -85,B 0,C 180,E1 25828.718,E2 25828.718} C_VEL
LIN {X 0,Y 535.912,Z 1003.561,A -85,B 0,C 180,E1 25826.471,E2 25826.471} C_VEL
LIN {X 0,Y 535.928,Z 1000.428,A -85,B 0,C 180,E1 25824.219,E2 25824.219} C_VEL
LIN {X 0,Y 535.971,Z 995.639,A -85,B 0,C 180,E1 25821.958,E2 25821.958} C_VEL
LIN {X 0,Y 536.054,Z 989.181,A -85,B 0,C 180,E1 25819.686,E2 25819.686} C_VEL
LIN {X 0,Y 536.207,Z 981.436,A -85,B 0,C 180,E1 25817.51,E2 25817.51} C_VEL
LIN {X 0,Y 536.456,Z 971.752,A -85,B 0,C 180,E1 25815.311,E2 25815.311} C_VEL
LIN {X 0,Y 536.835,Z 960.204,A -85,B 0,C 180,E1 25813.111,E2 25813.111} C_VEL
LIN {X 0,Y 537.319,Z 947.888,A -85,B 0,C 180,E1 25811.11,E2 25811.11} C_VEL
LIN {X 0,Y 537.958,Z 933.341,A -85,B 0,C 180,E1 25809.095,E2 25809.095} C_VEL
LIN {X 0,Y 538.675,Z 918.19,A -85,B 0,C 180,E1 25807.292,E2 25807.292} C_VEL
LIN {X 0,Y 539.593,Z 900.521,A -85,B 0,C 180,E1 25805.479,E2 25805.479} C_VEL
LIN {X 0,Y 540.509,Z 883.306,A -85,B 0,C 180,E1 25803.961,E2 25803.961} C_VEL
LIN {X 0,Y 541.433,Z 864.75,A -85,B 0,C 180,E1 25802.568,E2 25802.568} C_VEL
LIN {X 0,Y 542.403,Z 844.914,A -85,B 0,C 180,E1 25801.311,E2 25801.311} C_VEL
LIN {X 0,Y 543.297,Z 825.224,A -85,B 0,C 180,E1 25800.27,E2 25800.27} C_VEL
LIN {X 0,Y 544.071,Z 805.577,A -85,B 0,C 180,E1 25799.434,E2 25799.434} C_VEL
LIN {X 0,Y 544.767,Z 783.008,A -85,B 0,C 180,E1 25798.684,E2 25798.684} C_VEL
LIN {X 0,Y 545.351,Z 761.419,A -85,B 0,C 180,E1 25798.172,E2 25798.172} C_VEL
LIN {X 0,Y 547.014,Z 583.511,A -85,B 0,C 180,E1 25795.515,E2 25795.515} C_VEL
LIN {X 0,Y 547.985,Z 465.682,A -85,B 0,C 180,E1 25793.731,E2 25793.731} C_VEL
LIN {X 0,Y 546.341,Z 453.868,A -85,B 0,C 180,E1 25793.377,E2 25793.377} C_VEL
LIN {X 0,Y 547.98,Z 401.557,A -85,B 0,C 180,E1 25790.248,E2 25790.248} C_VEL
LIN {X 0,Y 548.247,Z 389.018,A -85,B 0,C 180,E1 25789.508,E2 25789.508} C_VEL
LIN {X 0,Y 536.503,Z 364.449,A -85,B 0,C 180,E1 25786.998,E2 25786.998} C_VEL
LIN {X 0,Y 536.443,Z 363.897,A -85,B 0,C 180,E1 25786.699,E2 25786.699} C_VEL
LIN {X 0,Y 536.399,Z 363.908,A -85,B 0,C 180,E1 25783.374,E2 25783.374} C_VEL
LIN {X 0,Y 536.465,Z 363.895,A -85,B 0,C 180,E1 25780.156,E2 25780.156} C_VEL
LIN {X 0,Y 536.4,Z 363.913,A -85,B 0,C 180,E1 25776.885,E2 25776.885} C_VEL
LIN {X 0,Y 536.403,Z 363.917,A -85,B 0,C 180,E1 25773.386,E2 25773.386} C_VEL
LIN {X 0,Y 536.432,Z 363.896,A -85,B 0,C 180,E1 25770.215,E2 25770.215} C_VEL
LIN {X 0,Y 536.387,Z 363.916,A -85,B 0,C 180,E1 25766.934,E2 25766.934} C_VEL
LIN {X 0,Y 536.447,Z 363.895,A -85,B 0,C 180,E1 25763.623,E2 25763.623} C_VEL
LIN {X 0,Y 536.386,Z 363.917,A -85,B 0,C 180,E1 25760.4,E2 25760.4} C_VEL
LIN {X 0,Y 536.388,Z 363.917,A -85,B 0,C 180,E1 25756.905,E2 25756.905} C_VEL
LIN {X 0,Y 536.414,Z 363.914,A -85,B 0,C 180,E1 25753.803,E2 25753.803} C_VEL
LIN {X 0,Y 536.381,Z 363.914,A -85,B 0,C 180,E1 25750.526,E2 25750.526} C_VEL
LIN {X 0,Y 536.462,Z 363.908,A -85,B 0,C 180,E1 25747.281,E2 25747.281} C_VEL
LIN {X 0,Y 536.387,Z 363.915,A -85,B 0,C 180,E1 25744.062,E2 25744.062} C_VEL
LIN {X 0,Y 536.426,Z 363.914,A -85,B 0,C 180,E1 25740.747,E2 25740.747} C_VEL
LIN {X 0,Y 536.402,Z 363.909,A -85,B 0,C 180,E1 25737.649,E2 25737.649} C_VEL
LIN {X 0,Y 536.402,Z 363.906,A -85,B 0,C 180,E1 25734.223,E2 25734.223} C_VEL
LIN {X 0,Y 536.45,Z 363.914,A -85,B 0,C 180,E1 25731.015,E2 25731.015} C_VEL
LIN {X 0,Y 536.401,Z 363.913,A -85,B 0,C 180,E1 25727.731,E2 25727.731} C_VEL
LIN {X 0,Y 536.456,Z 363.911,A -85,B 0,C 180,E1 25724.431,E2 25724.431} C_VEL
LIN {X 0,Y 536.415,Z 363.912,A -85,B 0,C 180,E1 25721.188,E2 25721.188} C_VEL
LIN {X 0,Y 536.416,Z 363.91,A -85,B 0,C 180,E1 25717.766,E2 25717.766} C_VEL
LIN {X 0,Y 536.46,Z 363.913,A -85,B 0,C 180,E1 25714.498,E2 25714.498} C_VEL
LIN {X 0,Y 536.413,Z 363.913,A -85,B 0,C 180,E1 25711.16,E2 25711.16} C_VEL
LIN {X 0,Y 536.461,Z 363.91,A -85,B 0,C 180,E1 25707.914,E2 25707.914} C_VEL
LIN {X 0,Y 536.422,Z 363.91,A -85,B 0,C 180,E1 25705.331,E2 25705.331} C_VEL
LIN {X 0,Y 535.431,Z 364.041,A -85,B 0,C 180,E1 25704.508,E2 25704.508} C_VEL
LIN {X 0,Y 528.978,Z 364.827,A -85,B 0,C 180,E1 25702.137,E2 25702.137} C_VEL
LIN {X 0,Y 528.51,Z 364.876,A -85,B 0,C 180,E1 25701.595,E2 25701.595} C_VEL
LIN {X 0,Y 528.52,Z 364.904,A -85,B 0,C 180,E1 25698.184,E2 25698.184} C_VEL
LIN {X 0,Y 528.485,Z 364.892,A -85,B 0,C 180,E1 25694.807,E2 25694.807} C_VEL
LIN {X 0,Y 528.527,Z 364.88,A -85,B 0,C 180,E1 25691.456,E2 25691.456} C_VEL
LIN {X 0,Y 528.511,Z 364.89,A -85,B 0,C 180,E1 25688.073,E2 25688.073} C_VEL
LIN {X 0,Y 528.492,Z 364.89,A -85,B 0,C 180,E1 25684.615,E2 25684.615} C_VEL
LIN {X 0,Y 528.549,Z 365.266,A -85,B 0,C 180,E1 25684.31,E2 25684.31} C_VEL
LIN {X 0,Y 533.761,Z 379.386,A -85,B 0,C 180,E1 25682.436,E2 25682.436} C_VEL
LIN {X 0,Y 535.511,Z 384.637,A -85,B 0,C 180,E1 25681.838,E2 25681.838} C_VEL
LIN {X 0,Y 538.295,Z 398.748,A -85,B 0,C 180,E1 25681.398,E2 25681.398} C_VEL
LIN {X 0,Y 536.147,Z 615.394,A -85,B 0,C 180,E1 25678.204,E2 25678.204} C_VEL
LIN {X 0,Y 535.77,Z 646.835,A -85,B 0,C 180,E1 25677.705,E2 25677.705} C_VEL
LIN {X 0,Y 535.269,Z 667.422,A -85,B 0,C 180,E1 25677.183,E2 25677.183} C_VEL
LIN {X 0,Y 534.586,Z 687.677,A -85,B 0,C 180,E1 25676.459,E2 25676.459} C_VEL
LIN {X 0,Y 533.833,Z 706.693,A -85,B 0,C 180,E1 25675.574,E2 25675.574} C_VEL
LIN {X 0,Y 532.97,Z 725.49,A -85,B 0,C 180,E1 25674.491,E2 25674.491} C_VEL
LIN {X 0,Y 532.067,Z 744.149,A -85,B 0,C 180,E1 25673.182,E2 25673.182} C_VEL
LIN {X 0,Y 531.225,Z 761.057,A -85,B 0,C 180,E1 25671.762,E2 25671.762} C_VEL
LIN {X 0,Y 530.44,Z 777.036,A -85,B 0,C 180,E1 25670.176,E2 25670.176} C_VEL
LIN {X 0,Y 529.742,Z 791.516,A -85,B 0,C 180,E1 25668.485,E2 25668.485} C_VEL
LIN {X 0,Y 529.137,Z 805.327,A -85,B 0,C 180,E1 25666.576,E2 25666.576} C_VEL
LIN {X 0,Y 528.68,Z 816.904,A -85,B 0,C 180,E1 25664.678,E2 25664.678} C_VEL
LIN {X 0,Y 528.359,Z 827.15,A -85,B 0,C 180,E1 25662.679,E2 25662.679} C_VEL
LIN {X 0,Y 528.134,Z 836.003,A -85,B 0,C 180,E1 25660.58,E2 25660.58} C_VEL
LIN {X 0,Y 528.015,Z 843.072,A -85,B 0,C 180,E1 25658.493,E2 25658.493} C_VEL
LIN {X 0,Y 527.944,Z 848.907,A -85,B 0,C 180,E1 25656.196,E2 25656.196} C_VEL
LIN {X 0,Y 527.92,Z 852.68,A -85,B 0,C 180,E1 25654.018,E2 25654.018} C_VEL
LIN {X 0,Y 527.912,Z 854.847,A -85,B 0,C 180,E1 25651.845,E2 25651.845} C_VEL
LIN {X 0,Y 527.903,Z 855.449,A -85,B 0,C 180,E1 25649.674,E2 25649.674} C_VEL
LIN {X 0,Y 527.905,Z 854.491,A -85,B 0,C 180,E1 25647.503,E2 25647.503} C_VEL
LIN {X 0,Y 527.92,Z 851.856,A -85,B 0,C 180,E1 25645.329,E2 25645.329} C_VEL
LIN {X 0,Y 527.952,Z 847.597,A -85,B 0,C 180,E1 25643.148,E2 25643.148} C_VEL
LIN {X 0,Y 528.021,Z 841.62,A -85,B 0,C 180,E1 25640.958,E2 25640.958} C_VEL
LIN {X 0,Y 528.166,Z 834.245,A -85,B 0,C 180,E1 25638.867,E2 25638.867} C_VEL
LIN {X 0,Y 528.425,Z 824.975,A -85,B 0,C 180,E1 25636.766,E2 25636.766} C_VEL
LIN {X 0,Y 528.781,Z 814.224,A -85,B 0,C 180,E1 25634.763,E2 25634.763} C_VEL
LIN {X 0,Y 529.256,Z 802.083,A -85,B 0,C 180,E1 25632.861,E2 25632.861} C_VEL
LIN {X 0,Y 529.901,Z 787.756,A -85,B 0,C 180,E1 25630.967,E2 25630.967} C_VEL
LIN {X 0,Y 530.673,Z 771.841,A -85,B 0,C 180,E1 25629.193,E2 25629.193} C_VEL
LIN {X 0,Y 531.517,Z 755.095,A -85,B 0,C 180,E1 25627.62,E2 25627.62} C_VEL
LIN {X 0,Y 532.404,Z 737.724,A -85,B 0,C 180,E1 25626.247,E2 25626.247} C_VEL
LIN {X 0,Y 533.264,Z 719.596,A -85,B 0,C 180,E1 25625.05,E2 25625.05} C_VEL
LIN {X 0,Y 534.082,Z 700.469,A -85,B 0,C 180,E1 25624.021,E2 25624.021} C_VEL
LIN {X 0,Y 534.819,Z 681.015,A -85,B 0,C 180,E1 25623.193,E2 25623.193} C_VEL
LIN {X 0,Y 535.427,Z 660.75,A -85,B 0,C 180,E1 25622.539,E2 25622.539} C_VEL
LIN {X 0,Y 535.894,Z 639.535,A -85,B 0,C 180,E1 25622.069,E2 25622.069} C_VEL
LIN {X 0,Y 538.227,Z 406.759,A -85,B 0,C 180,E1 25618.627,E2 25618.627} C_VEL
LIN {X 0,Y 538.117,Z 396.715,A -85,B 0,C 180,E1 25618.46,E2 25618.46} C_VEL
LIN {X 0,Y 535.411,Z 384.368,A -85,B 0,C 180,E1 25618.052,E2 25618.052} C_VEL
LIN {X 0,Y 530.926,Z 371.384,A -85,B 0,C 180,E1 25616.443,E2 25616.443} C_VEL
LIN {X 0,Y 528.524,Z 365.089,A -85,B 0,C 180,E1 25615.556,E2 25615.556} C_VEL
LIN {X 0,Y 528.523,Z 364.884,A -85,B 0,C 180,E1 25612.201,E2 25612.201} C_VEL
LIN {X 0,Y 528.508,Z 364.881,A -85,B 0,C 180,E1 25608.829,E2 25608.829} C_VEL
LIN {X 0,Y 528.493,Z 364.893,A -85,B 0,C 180,E1 25605.346,E2 25605.346} C_VEL
LIN {X 0,Y 528.523,Z 364.901,A -85,B 0,C 180,E1 25601.898,E2 25601.898} C_VEL
LIN {X 0,Y 528.505,Z 364.876,A -85,B 0,C 180,E1 25598.494,E2 25598.494} C_VEL
LIN {X 0,Y 528.487,Z 364.901,A -85,B 0,C 180,E1 25595.11,E2 25595.11} C_VEL
LIN {X 0,Y 528.528,Z 364.902,A -85,B 0,C 180,E1 25591.73,E2 25591.73} C_VEL
LIN {X 0,Y 528.486,Z 364.9,A -85,B 0,C 180,E1 25588.398,E2 25588.398} C_VEL
LIN {X 0,Y 528.485,Z 364.902,A -85,B 0,C 180,E1 25584.955,E2 25584.955} C_VEL
LIN {X 0,Y 528.528,Z 364.896,A -85,B 0,C 180,E1 25581.648,E2 25581.648} C_VEL
LIN {X 0,Y 528.472,Z 364.898,A -85,B 0,C 180,E1 25578.305,E2 25578.305} C_VEL
LIN {X 0,Y 528.496,Z 364.898,A -85,B 0,C 180,E1 25574.91,E2 25574.91} C_VEL
LIN {X 0,Y 528.491,Z 364.901,A -85,B 0,C 180,E1 25571.68,E2 25571.68} C_VEL
LIN {X 0,Y 528.464,Z 364.903,A -85,B 0,C 180,E1 25568.268,E2 25568.268} C_VEL
LIN {X 0,Y 528.521,Z 364.897,A -85,B 0,C 180,E1 25564.993,E2 25564.993} C_VEL
LIN {X 0,Y 528.459,Z 364.897,A -85,B 0,C 180,E1 25561.735,E2 25561.735} C_VEL
LIN {X 0,Y 528.466,Z 364.9,A -85,B 0,C 180,E1 25558.266,E2 25558.266} C_VEL
LIN {X 0,Y 528.499,Z 364.903,A -85,B 0,C 180,E1 25555.008,E2 25555.008} C_VEL
LIN {X 0,Y 528.447,Z 364.904,A -85,B 0,C 180,E1 25551.733,E2 25551.733} C_VEL
LIN {X 0,Y 528.503,Z 364.899,A -85,B 0,C 180,E1 25548.432,E2 25548.432} C_VEL
LIN {X 0,Y 528.446,Z 364.903,A -85,B 0,C 180,E1 25545.201,E2 25545.201} C_VEL
LIN {X 0,Y 528.446,Z 364.902,A -85,B 0,C 180,E1 25541.695,E2 25541.695} C_VEL
LIN {X 0,Y 528.498,Z 364.905,A -85,B 0,C 180,E1 25538.468,E2 25538.468} C_VEL
LIN {X 0,Y 528.441,Z 364.889,A -85,B 0,C 180,E1 25535.163,E2 25535.163} C_VEL
LIN {X 0,Y 528.49,Z 364.9,A -85,B 0,C 180,E1 25531.83,E2 25531.83} C_VEL
LIN {X 0,Y 528.453,Z 364.891,A -85,B 0,C 180,E1 25528.774,E2 25528.774} C_VEL
LIN {X 0,Y 528.463,Z 364.894,A -85,B 0,C 180,E1 25525.285,E2 25525.285} C_VEL
LIN {X 0,Y 528.506,Z 364.905,A -85,B 0,C 180,E1 25522.059,E2 25522.059} C_VEL
LIN {X 0,Y 528.459,Z 364.9,A -85,B 0,C 180,E1 25518.821,E2 25518.821} C_VEL
LIN {X 0,Y 528.516,Z 364.884,A -85,B 0,C 180,E1 25515.492,E2 25515.492} C_VEL
LIN {X 0,Y 528.553,Z 365.106,A -85,B 0,C 180,E1 25513.686,E2 25513.686} C_VEL
LIN {X 0,Y 529.211,Z 367.294,A -85,B 0,C 180,E1 25513.419,E2 25513.419} C_VEL
LIN {X 0,Y 541.449,Z 392.679,A -85,B 0,C 180,E1 25510.789,E2 25510.789} C_VEL
LIN {X 0,Y 540.027,Z 443.692,A -85,B 0,C 180,E1 25507.76,E2 25507.76} C_VEL
LIN {X 0,Y 539.777,Z 455.305,A -85,B 0,C 180,E1 25507.087,E2 25507.087} C_VEL
LIN {X 0,Y 541.676,Z 469.531,A -85,B 0,C 180,E1 25506.698,E2 25506.698} C_VEL
LIN {X 0,Y 539.296,Z 694.718,A -85,B 0,C 180,E1 25503.296,E2 25503.296} C_VEL
LIN {X 0,Y 538.534,Z 762.511,A -85,B 0,C 180,E1 25502.258,E2 25502.258} C_VEL
LIN {X 0,Y 537.872,Z 784.135,A -85,B 0,C 180,E1 25501.73,E2 25501.73} C_VEL
LIN {X 0,Y 537.095,Z 806.286,A -85,B 0,C 180,E1 25500.977,E2 25500.977} C_VEL
LIN {X 0,Y 536.2,Z 826.651,A -85,B 0,C 180,E1 25500.092,E2 25500.092} C_VEL
LIN {X 0,Y 535.175,Z 846.699,A -85,B 0,C 180,E1 25499.004,E2 25499.004} C_VEL
LIN {X 0,Y 534.038,Z 867.166,A -85,B 0,C 180,E1 25497.664,E2 25497.664} C_VEL
LIN {X 0,Y 532.932,Z 886.465,A -85,B 0,C 180,E1 25496.159,E2 25496.159} C_VEL
LIN {X 0,Y 531.903,Z 904.362,A -85,B 0,C 180,E1 25494.521,E2 25494.521} C_VEL
LIN {X 0,Y 530.934,Z 920.714,A -85,B 0,C 180,E1 25492.766,E2 25492.766} C_VEL
LIN {X 0,Y 530.108,Z 935.886,A -85,B 0,C 180,E1 25490.882,E2 25490.882} C_VEL
LIN {X 0,Y 529.417,Z 950.057,A -85,B 0,C 180,E1 25488.84,E2 25488.84} C_VEL
LIN {X 0,Y 528.877,Z 962.737,A -85,B 0,C 180,E1 25486.699,E2 25486.699} C_VEL
LIN {X 0,Y 528.483,Z 973.337,A -85,B 0,C 180,E1 25484.573,E2 25484.573} C_VEL
LIN {X 0,Y 528.197,Z 983.074,A -85,B 0,C 180,E1 25482.239,E2 25482.239} C_VEL
LIN {X 0,Y 528.04,Z 990.591,A -85,B 0,C 180,E1 25480.032,E2 25480.032} C_VEL
LIN {X 0,Y 527.95,Z 996.654,A -85,B 0,C 180,E1 25477.727,E2 25477.727} C_VEL
LIN {X 0,Y 527.914,Z 1001.144,A -85,B 0,C 180,E1 25475.434,E2 25475.434} C_VEL
LIN {X 0,Y 527.908,Z 1003.898,A -85,B 0,C 180,E1 25473.257,E2 25473.257} C_VEL
LIN {X 0,Y 527.901,Z 1005.328,A -85,B 0,C 180,E1 25470.868,E2 25470.868} C_VEL
LIN {X 0,Y 527.903,Z 1005.209,A -85,B 0,C 180,E1 25468.59,E2 25468.59} C_VEL
LIN {X 0,Y 527.909,Z 1003.448,A -85,B 0,C 180,E1 25466.309,E2 25466.309} C_VEL
LIN {X 0,Y 527.933,Z 999.952,A -85,B 0,C 180,E1 25463.878,E2 25463.878} C_VEL
LIN {X 0,Y 527.988,Z 994.875,A -85,B 0,C 180,E1 25461.507,E2 25461.507} C_VEL
LIN {X 0,Y 528.09,Z 988.117,A -85,B 0,C 180,E1 25459.198,E2 25459.198} C_VEL
LIN {X 0,Y 528.294,Z 979.605,A -85,B 0,C 180,E1 25456.875,E2 25456.875} C_VEL
LIN {X 0,Y 528.617,Z 969.696,A -85,B 0,C 180,E1 25454.647,E2 25454.647} C_VEL
LIN {X 0,Y 529.053,Z 958.286,A -85,B 0,C 180,E1 25452.515,E2 25452.515} C_VEL
LIN {X 0,Y 529.665,Z 944.805,A -85,B 0,C 180,E1 25450.368,E2 25450.368} C_VEL
LIN {X 0,Y 530.401,Z 930.674,A -85,B 0,C 180,E1 25448.435,E2 25448.435} C_VEL
LIN {X 0,Y 531.29,Z 914.839,A -85,B 0,C 180,E1 25446.571,E2 25446.571} C_VEL
LIN {X 0,Y 532.239,Z 898.089,A -85,B 0,C 180,E1 25444.88,E2 25444.88} C_VEL
LIN {X 0,Y 533.335,Z 879.437,A -85,B 0,C 180,E1 25443.264,E2 25443.264} C_VEL
LIN {X 0,Y 534.442,Z 860.594,A -85,B 0,C 180,E1 25441.875,E2 25441.875} C_VEL
LIN {X 0,Y 535.459,Z 840.895,A -85,B 0,C 180,E1 25440.658,E2 25440.658} C_VEL
LIN {X 0,Y 536.461,Z 821.016,A -85,B 0,C 180,E1 25439.648,E2 25439.648} C_VEL
LIN {X 0,Y 537.336,Z 800.48,A -85,B 0,C 180,E1 25438.799,E2 25438.799} C_VEL
LIN {X 0,Y 538.049,Z 779.362,A -85,B 0,C 180,E1 25438.138,E2 25438.138} C_VEL
LIN {X 0,Y 538.605,Z 756.886,A -85,B 0,C 180,E1 25437.643,E2 25437.643} C_VEL
LIN {X 0,Y 540.904,Z 539.306,A -85,B 0,C 180,E1 25434.365,E2 25434.365} C_VEL
LIN {X 0,Y 541.512,Z 466.977,A -85,B 0,C 180,E1 25433.247,E2 25433.247} C_VEL
LIN {X 0,Y 539.693,Z 453.868,A -85,B 0,C 180,E1 25432.851,E2 25432.851} C_VEL
LIN {X 0,Y 540.997,Z 410.07,A -85,B 0,C 180,E1 25430.25,E2 25430.25} C_VEL
LIN {X 0,Y 541.327,Z 392.202,A -85,B 0,C 180,E1 25429.173,E2 25429.173} C_VEL
LIN {X 0,Y 528.612,Z 365.427,A -85,B 0,C 180,E1 25426.379,E2 25426.379} C_VEL
LIN {X 0,Y 528.506,Z 364.895,A -85,B 0,C 180,E1 25426.12,E2 25426.12} C_VEL
LIN {X 0,Y 528.471,Z 364.9,A -85,B 0,C 180,E1 25422.93,E2 25422.93} C_VEL
LIN {X 0,Y 528.463,Z 364.895,A -85,B 0,C 180,E1 25419.473,E2 25419.473} C_VEL
LIN {X 0,Y 528.505,Z 364.887,A -85,B 0,C 180,E1 25416.308,E2 25416.308} C_VEL
LIN {X 0,Y 528.454,Z 364.906,A -85,B 0,C 180,E1 25413.018,E2 25413.018} C_VEL
LIN {X 0,Y 528.502,Z 364.885,A -85,B 0,C 180,E1 25409.714,E2 25409.714} C_VEL
LIN {X 0,Y 528.456,Z 364.905,A -85,B 0,C 180,E1 25406.513,E2 25406.513} C_VEL
LIN {X 0,Y 528.452,Z 364.898,A -85,B 0,C 180,E1 25403.057,E2 25403.057} C_VEL
LIN {X 0,Y 528.486,Z 364.906,A -85,B 0,C 180,E1 25399.91,E2 25399.91} C_VEL
LIN {X 0,Y 528.438,Z 364.906,A -85,B 0,C 180,E1 25396.601,E2 25396.601} C_VEL
LIN {X 0,Y 528.503,Z 364.905,A -85,B 0,C 180,E1 25393.344,E2 25393.344} C_VEL
LIN {X 0,Y 528.447,Z 364.903,A -85,B 0,C 180,E1 25390.134,E2 25390.134} C_VEL
LIN {X 0,Y 528.456,Z 364.902,A -85,B 0,C 180,E1 25386.627,E2 25386.627} C_VEL
LIN {X 0,Y 528.489,Z 364.903,A -85,B 0,C 180,E1 25383.471,E2 25383.471} C_VEL
LIN {X 0,Y 528.452,Z 364.904,A -85,B 0,C 180,E1 25380.217,E2 25380.217} C_VEL
LIN {X 0,Y 528.518,Z 364.902,A -85,B 0,C 180,E1 25376.963,E2 25376.963} C_VEL
LIN {X 0,Y 528.458,Z 364.896,A -85,B 0,C 180,E1 25373.7,E2 25373.7} C_VEL
LIN {X 0,Y 528.478,Z 364.896,A -85,B 0,C 180,E1 25370.266,E2 25370.266} C_VEL
LIN {X 0,Y 528.505,Z 364.904,A -85,B 0,C 180,E1 25366.989,E2 25366.989} C_VEL
LIN {X 0,Y 528.464,Z 364.902,A -85,B 0,C 180,E1 25363.626,E2 25363.626} C_VEL
LIN {X 0,Y 528.518,Z 364.899,A -85,B 0,C 180,E1 25360.321,E2 25360.321} C_VEL
LIN {X 0,Y 528.479,Z 364.901,A -85,B 0,C 180,E1 25357.061,E2 25357.061} C_VEL
LIN {X 0,Y 528.478,Z 364.898,A -85,B 0,C 180,E1 25353.601,E2 25353.601} C_VEL
LIN {X 0,Y 528.529,Z 364.896,A -85,B 0,C 180,E1 25350.254,E2 25350.254} C_VEL
LIN {X 0,Y 528.481,Z 364.903,A -85,B 0,C 180,E1 25346.934,E2 25346.934} C_VEL
LIN {X 0,Y 528.498,Z 364.898,A -85,B 0,C 180,E1 25343.51,E2 25343.51} C_VEL
LIN {X 0,Y 528.51,Z 364.876,A -85,B 0,C 180,E1 25341.595,E2 25341.595} C_VEL
LIN {X 0,Y 527.483,Z 365.007,A -85,B 0,C 180,E1 25340.76,E2 25340.76} C_VEL
LIN {X 0,Y 521.12,Z 365.826,A -85,B 0,C 180,E1 25338.414,E2 25338.414} C_VEL
LIN {X 0,Y 520.587,Z 365.885,A -85,B 0,C 180,E1 25337.803,E2 25337.803} C_VEL
LIN {X 0,Y 520.56,Z 365.883,A -85,B 0,C 180,E1 25334.352,E2 25334.352} C_VEL
LIN {X 0,Y 520.55,Z 365.872,A -85,B 0,C 180,E1 25330.818,E2 25330.818} C_VEL
LIN {X 0,Y 520.583,Z 365.869,A -85,B 0,C 180,E1 25327.501,E2 25327.501} C_VEL
LIN {X 0,Y 520.607,Z 366.145,A -85,B 0,C 180,E1 25324.957,E2 25324.957} C_VEL
LIN {X 0,Y 526.49,Z 381.766,A -85,B 0,C 180,E1 25322.822,E2 25322.822} C_VEL
LIN {X 0,Y 527.8,Z 385.422,A -85,B 0,C 180,E1 25322.415,E2 25322.415} C_VEL
LIN {X 0,Y 529.715,Z 389.446,A -85,B 0,C 180,E1 25322.198,E2 25322.198} C_VEL
LIN {X 0,Y 531.712,Z 400.319,A -85,B 0,C 180,E1 25321.868,E2 25321.868} C_VEL
LIN {X 0,Y 529.055,Z 629.214,A -85,B 0,C 180,E1 25318.43,E2 25318.43} C_VEL
LIN {X 0,Y 528.593,Z 651.704,A -85,B 0,C 180,E1 25318.011,E2 25318.011} C_VEL
LIN {X 0,Y 527.949,Z 672.228,A -85,B 0,C 180,E1 25317.424,E2 25317.424} C_VEL
LIN {X 0,Y 527.185,Z 692.32,A -85,B 0,C 180,E1 25316.647,E2 25316.647} C_VEL
LIN {X 0,Y 526.335,Z 711.077,A -85,B 0,C 180,E1 25315.723,E2 25315.723} C_VEL
LIN {X 0,Y 525.388,Z 729.983,A -85,B 0,C 180,E1 25314.568,E2 25314.568} C_VEL
LIN {X 0,Y 524.38,Z 748.223,A -85,B 0,C 180,E1 25313.212,E2 25313.212} C_VEL
LIN {X 0,Y 523.43,Z 764.706,A -85,B 0,C 180,E1 25311.749,E2 25311.749} C_VEL
LIN {X 0,Y 522.554,Z 780.581,A -85,B 0,C 180,E1 25310.085,E2 25310.085} C_VEL
LIN {X 0,Y 521.798,Z 794.94,A -85,B 0,C 180,E1 25308.313,E2 25308.313} C_VEL
LIN {X 0,Y 521.16,Z 808.224,A -85,B 0,C 180,E1 25306.379,E2 25306.379} C_VEL
LIN {X 0,Y 520.674,Z 819.975,A -85,B 0,C 180,E1 25304.341,E2 25304.341} C_VEL
LIN {X 0,Y 520.323,Z 830.205,A -85,B 0,C 180,E1 25302.201,E2 25302.201} C_VEL
LIN {X 0,Y 520.102,Z 838.429,A -85,B 0,C 180,E1 25300.074,E2 25300.074} C_VEL
LIN {X 0,Y 519.992,Z 844.888,A -85,B 0,C 180,E1 25297.957,E2 25297.957} C_VEL
LIN {X 0,Y 519.934,Z 849.972,A -85,B 0,C 180,E1 25295.738,E2 25295.738} C_VEL
LIN {X 0,Y 519.907,Z 853.408,A -85,B 0,C 180,E1 25293.515,E2 25293.515} C_VEL
LIN {X 0,Y 519.901,Z 855.182,A -85,B 0,C 180,E1 25291.322,E2 25291.322} C_VEL
LIN {X 0,Y 519.909,Z 855.336,A -85,B 0,C 180,E1 25289.118,E2 25289.118} C_VEL
LIN {X 0,Y 519.905,Z 853.827,A -85,B 0,C 180,E1 25286.803,E2 25286.803} C_VEL
LIN {X 0,Y 519.915,Z 850.758,A -85,B 0,C 180,E1 25284.593,E2 25284.593} C_VEL
LIN {X 0,Y 519.971,Z 846.041,A -85,B 0,C 180,E1 25282.376,E2 25282.376} C_VEL
LIN {X 0,Y 520.087,Z 839.496,A -85,B 0,C 180,E1 25280.149,E2 25280.149} C_VEL
LIN {X 0,Y 520.277,Z 831.446,A -85,B 0,C 180,E1 25278.012,E2 25278.012} C_VEL
LIN {X 0,Y 520.603,Z 821.571,A -85,B 0,C 180,E1 25275.883,E2 25275.883} C_VEL
LIN {X 0,Y 521.071,Z 810.165,A -85,B 0,C 180,E1 25273.846,E2 25273.846} C_VEL
LIN {X 0,Y 521.676,Z 797.374,A -85,B 0,C 180,E1 25271.925,E2 25271.925} C_VEL
LIN {X 0,Y 522.413,Z 783.492,A -85,B 0,C 180,E1 25270.154,E2 25270.154} C_VEL
LIN {X 0,Y 523.304,Z 767.436,A -85,B 0,C 180,E1 25268.422,E2 25268.422} C_VEL
LIN {X 0,Y 524.267,Z 750.29,A -85,B 0,C 180,E1 25266.869,E2 25266.869} C_VEL
LIN {X 0,Y 525.214,Z 732.828,A -85,B 0,C 180,E1 25265.542,E2 25265.542} C_VEL
LIN {X 0,Y 526.149,Z 714.561,A -85,B 0,C 180,E1 25264.387,E2 25264.387} C_VEL
LIN {X 0,Y 527.048,Z 695.486,A -85,B 0,C 180,E1 25263.405,E2 25263.405} C_VEL
LIN {X 0,Y 527.813,Z 675.932,A -85,B 0,C 180,E1 25262.61,E2 25262.61} C_VEL
LIN {X 0,Y 528.532,Z 654.759,A -85,B 0,C 180,E1 25261.973,E2 25261.973} C_VEL
LIN {X 0,Y 528.996,Z 634.029,A -85,B 0,C 180,E1 25261.554,E2 25261.554} C_VEL
LIN {X 0,Y 531.709,Z 403.444,A -85,B 0,C 180,E1 25258.083,E2 25258.083} C_VEL
LIN {X 0,Y 531.505,Z 398.083,A -85,B 0,C 180,E1 25257.984,E2 25257.984} C_VEL
LIN {X 0,Y 529.208,Z 388.056,A -85,B 0,C 180,E1 25257.648,E2 25257.648} C_VEL
LIN {X 0,Y 527.404,Z 384.537,A -85,B 0,C 180,E1 25257.428,E2 25257.428} C_VEL
LIN {X 0,Y 523.066,Z 372.518,A -85,B 0,C 180,E1 25255.863,E2 25255.863} C_VEL
LIN {X 0,Y 520.616,Z 366.156,A -85,B 0,C 180,E1 25254.957,E2 25254.957} C_VEL
LIN {X 0,Y 520.58,Z 365.874,A -85,B 0,C 180,E1 25251.95,E2 25251.95} C_VEL
LIN {X 0,Y 520.587,Z 365.867,A -85,B 0,C 180,E1 25248.505,E2 25248.505} C_VEL
LIN {X 0,Y 520.551,Z 365.88,A -85,B 0,C 180,E1 25245.135,E2 25245.135} C_VEL
LIN {X 0,Y 520.576,Z 365.894,A -85,B 0,C 180,E1 25241.648,E2 25241.648} C_VEL
LIN {X 0,Y 520.584,Z 365.863,A -85,B 0,C 180,E1 25238.203,E2 25238.203} C_VEL
LIN {X 0,Y 520.544,Z 365.888,A -85,B 0,C 180,E1 25234.784,E2 25234.784} C_VEL
LIN {X 0,Y 520.568,Z 365.887,A -85,B 0,C 180,E1 25231.367,E2 25231.367} C_VEL
LIN {X 0,Y 520.588,Z 365.887,A -85,B 0,C 180,E1 25227.944,E2 25227.944} C_VEL
LIN {X 0,Y 520.537,Z 365.889,A -85,B 0,C 180,E1 25224.513,E2 25224.513} C_VEL
LIN {X 0,Y 520.571,Z 365.892,A -85,B 0,C 180,E1 25221.167,E2 25221.167} C_VEL
LIN {X 0,Y 520.564,Z 365.885,A -85,B 0,C 180,E1 25217.782,E2 25217.782} C_VEL
LIN {X 0,Y 520.529,Z 365.888,A -85,B 0,C 180,E1 25214.461,E2 25214.461} C_VEL
LIN {X 0,Y 520.586,Z 365.886,A -85,B 0,C 180,E1 25211.186,E2 25211.186} C_VEL
LIN {X 0,Y 520.529,Z 365.891,A -85,B 0,C 180,E1 25207.839,E2 25207.839} C_VEL
LIN {X 0,Y 520.526,Z 365.893,A -85,B 0,C 180,E1 25204.297,E2 25204.297} C_VEL
LIN {X 0,Y 520.582,Z 365.883,A -85,B 0,C 180,E1 25200.991,E2 25200.991} C_VEL
LIN {X 0,Y 520.515,Z 365.888,A -85,B 0,C 180,E1 25197.688,E2 25197.688} C_VEL
LIN {X 0,Y 520.528,Z 365.891,A -85,B 0,C 180,E1 25194.216,E2 25194.216} C_VEL
LIN {X 0,Y 520.528,Z 365.892,A -85,B 0,C 180,E1 25191.161,E2 25191.161} C_VEL
LIN {X 0,Y 520.509,Z 365.894,A -85,B 0,C 180,E1 25187.802,E2 25187.802} C_VEL
LIN {X 0,Y 520.574,Z 365.886,A -85,B 0,C 180,E1 25184.516,E2 25184.516} C_VEL
LIN {X 0,Y 520.503,Z 365.891,A -85,B 0,C 180,E1 25181.173,E2 25181.173} C_VEL
LIN {X 0,Y 520.522,Z 365.886,A -85,B 0,C 180,E1 25177.765,E2 25177.765} C_VEL
LIN {X 0,Y 520.542,Z 365.877,A -85,B 0,C 180,E1 25174.514,E2 25174.514} C_VEL
LIN {X 0,Y 520.508,Z 365.89,A -85,B 0,C 180,E1 25171.147,E2 25171.147} C_VEL
LIN {X 0,Y 520.571,Z 365.886,A -85,B 0,C 180,E1 25167.857,E2 25167.857} C_VEL
LIN {X 0,Y 520.525,Z 365.876,A -85,B 0,C 180,E1 25164.525,E2 25164.525} C_VEL
LIN {X 0,Y 520.523,Z 365.89,A -85,B 0,C 180,E1 25161.067,E2 25161.067} C_VEL
LIN {X 0,Y 520.578,Z 365.894,A -85,B 0,C 180,E1 25157.843,E2 25157.843} C_VEL
LIN {X 0,Y 520.526,Z 365.9,A -85,B 0,C 180,E1 25154.511,E2 25154.511} C_VEL
LIN {X 0,Y 520.648,Z 366.562,A -85,B 0,C 180,E1 25154.249,E2 25154.249} C_VEL
LIN {X 0,Y 534.642,Z 396.358,A -85,B 0,C 180,E1 25151.091,E2 25151.091} C_VEL
LIN {X 0,Y 533.076,Z 449.984,A -85,B 0,C 180,E1 25147.895,E2 25147.895} C_VEL
LIN {X 0,Y 533.145,Z 455.709,A -85,B 0,C 180,E1 25147.6,E2 25147.6} C_VEL
LIN {X 0,Y 535.247,Z 470.849,A -85,B 0,C 180,E1 25147.191,E2 25147.191} C_VEL
LIN {X 0,Y 532.596,Z 696.113,A -85,B 0,C 180,E1 25143.749,E2 25143.749} C_VEL
LIN {X 0,Y 531.761,Z 762.695,A -85,B 0,C 180,E1 25142.716,E2 25142.716} C_VEL
LIN {X 0,Y 531.04,Z 784.263,A -85,B 0,C 180,E1 25142.182,E2 25142.182} C_VEL
LIN {X 0,Y 530.182,Z 806.282,A -85,B 0,C 180,E1 25141.426,E2 25141.426} C_VEL
LIN {X 0,Y 529.211,Z 826.438,A -85,B 0,C 180,E1 25140.543,E2 25140.543} C_VEL
LIN {X 0,Y 528.047,Z 846.853,A -85,B 0,C 180,E1 25139.424,E2 25139.424} C_VEL
LIN {X 0,Y 526.793,Z 867.162,A -85,B 0,C 180,E1 25138.077,E2 25138.077} C_VEL
LIN {X 0,Y 525.568,Z 886.462,A -85,B 0,C 180,E1 25136.553,E2 25136.553} C_VEL
LIN {X 0,Y 524.426,Z 904.136,A -85,B 0,C 180,E1 25134.918,E2 25134.918} C_VEL
LIN {X 0,Y 523.329,Z 920.714,A -85,B 0,C 180,E1 25133.116,E2 25133.116} C_VEL
LIN {X 0,Y 522.407,Z 935.884,A -85,B 0,C 180,E1 25131.205,E2 25131.205} C_VEL
LIN {X 0,Y 521.625,Z 950.059,A -85,B 0,C 180,E1 25129.132,E2 25129.132} C_VEL
LIN {X 0,Y 521.013,Z 962.736,A -85,B 0,C 180,E1 25126.958,E2 25126.958} C_VEL
LIN {X 0,Y 520.567,Z 973.336,A -85,B 0,C 180,E1 25124.799,E2 25124.799} C_VEL
LIN {X 0,Y 520.244,Z 983.074,A -85,B 0,C 180,E1 25122.429,E2 25122.429} C_VEL
LIN {X 0,Y 520.064,Z 990.708,A -85,B 0,C 180,E1 25120.15,E2 25120.15} C_VEL
LIN {X 0,Y 519.965,Z 996.654,A -85,B 0,C 180,E1 25117.847,E2 25117.847} C_VEL
LIN {X 0,Y 519.912,Z 1001.304,A -85,B 0,C 180,E1 25115.407,E2 25115.407} C_VEL
LIN {X 0,Y 519.905,Z 1004.011,A -85,B 0,C 180,E1 25113.197,E2 25113.197} C_VEL
LIN {X 0,Y 519.896,Z 1005.351,A -85,B 0,C 180,E1 25110.772,E2 25110.772} C_VEL
LIN {X 0,Y 519.899,Z 1005.15,A -85,B 0,C 180,E1 25108.458,E2 25108.458} C_VEL
LIN {X 0,Y 519.91,Z 1003.333,A -85,B 0,C 180,E1 25106.141,E2 25106.141} C_VEL
LIN {X 0,Y 519.938,Z 999.811,A -85,B 0,C 180,E1 25103.708,E2 25103.708} C_VEL
LIN {X 0,Y 519.992,Z 994.875,A -85,B 0,C 180,E1 25101.375,E2 25101.375} C_VEL
LIN {X 0,Y 520.115,Z 988.118,A -85,B 0,C 180,E1 25099.03,E2 25099.03} C_VEL
LIN {X 0,Y 520.349,Z 979.604,A -85,B 0,C 180,E1 25096.67,E2 25096.67} C_VEL
LIN {X 0,Y 520.718,Z 969.695,A -85,B 0,C 180,E1 25094.408,E2 25094.408} C_VEL
LIN {X 0,Y 521.213,Z 958.288,A -85,B 0,C 180,E1 25092.243,E2 25092.243} C_VEL
LIN {X 0,Y 521.903,Z 944.803,A -85,B 0,C 180,E1 25090.064,E2 25090.064} C_VEL
LIN {X 0,Y 522.734,Z 930.459,A -85,B 0,C 180,E1 25088.076,E2 25088.076} C_VEL
LIN {X 0,Y 523.739,Z 914.642,A -85,B 0,C 180,E1 25086.189,E2 25086.189} C_VEL
LIN {X 0,Y 524.831,Z 897.653,A -85,B 0,C 180,E1 25084.457,E2 25084.457} C_VEL
LIN {X 0,Y 526.043,Z 878.848,A -85,B 0,C 180,E1 25082.814,E2 25082.814} C_VEL
LIN {X 0,Y 527.293,Z 859.677,A -85,B 0,C 180,E1 25081.395,E2 25081.395} C_VEL
LIN {X 0,Y 528.382,Z 840.791,A -85,B 0,C 180,E1 25080.22,E2 25080.22} C_VEL
LIN {X 0,Y 529.52,Z 820.112,A -85,B 0,C 180,E1 25079.163,E2 25079.163} C_VEL
LIN {X 0,Y 530.486,Z 799.298,A -85,B 0,C 180,E1 25078.306,E2 25078.306} C_VEL
LIN {X 0,Y 531.263,Z 778.693,A -85,B 0,C 180,E1 25077.662,E2 25077.662} C_VEL
LIN {X 0,Y 531.852,Z 756.434,A -85,B 0,C 180,E1 25077.172,E2 25077.172} C_VEL
LIN {X 0,Y 534.393,Z 540.324,A -85,B 0,C 180,E1 25073.88,E2 25073.88} C_VEL
LIN {X 0,Y 535.094,Z 468.402,A -85,B 0,C 180,E1 25072.756,E2 25072.756} C_VEL
LIN {X 0,Y 533.002,Z 454.062,A -85,B 0,C 180,E1 25072.338,E2 25072.338} C_VEL
LIN {X 0,Y 534.506,Z 400.804,A -85,B 0,C 180,E1 25069.178,E2 25069.178} C_VEL
LIN {X 0,Y 534.446,Z 395.696,A -85,B 0,C 180,E1 25068.851,E2 25068.851} C_VEL
LIN {X 0,Y 521.926,Z 369.454,A -85,B 0,C 180,E1 25066.079,E2 25066.079} C_VEL
LIN {X 0,Y 520.575,Z 366.181,A -85,B 0,C 180,E1 25065.68,E2 25065.68} C_VEL
LIN {X 0,Y 520.548,Z 365.873,A -85,B 0,C 180,E1 25063.9,E2 25063.9} C_VEL
LIN {X 0,Y 520.551,Z 365.875,A -85,B 0,C 180,E1 25060.627,E2 25060.627} C_VEL
LIN {X 0,Y 520.519,Z 365.892,A -85,B 0,C 180,E1 25057.234,E2 25057.234} C_VEL
LIN {X 0,Y 520.569,Z 365.888,A -85,B 0,C 180,E1 25053.849,E2 25053.849} C_VEL
LIN {X 0,Y 520.52,Z 365.874,A -85,B 0,C 180,E1 25050.599,E2 25050.599} C_VEL
LIN {X 0,Y 520.514,Z 365.894,A -85,B 0,C 180,E1 25047.081,E2 25047.081} C_VEL
LIN {X 0,Y 520.572,Z 365.866,A -85,B 0,C 180,E1 25043.787,E2 25043.787} C_VEL
LIN {X 0,Y 520.505,Z 365.895,A -85,B 0,C 180,E1 25040.581,E2 25040.581} C_VEL
LIN {X 0,Y 520.535,Z 365.895,A -85,B 0,C 180,E1 25037.206,E2 25037.206} C_VEL
LIN {X 0,Y 520.518,Z 365.892,A -85,B 0,C 180,E1 25034.006,E2 25034.006} C_VEL
LIN {X 0,Y 520.507,Z 365.891,A -85,B 0,C 180,E1 25030.626,E2 25030.626} C_VEL
LIN {X 0,Y 520.584,Z 365.884,A -85,B 0,C 180,E1 25027.282,E2 25027.282} C_VEL
LIN {X 0,Y 520.513,Z 365.893,A -85,B 0,C 180,E1 25023.965,E2 25023.965} C_VEL
LIN {X 0,Y 520.523,Z 365.893,A -85,B 0,C 180,E1 25020.44,E2 25020.44} C_VEL
LIN {X 0,Y 520.571,Z 365.887,A -85,B 0,C 180,E1 25017.137,E2 25017.137} C_VEL
LIN {X 0,Y 520.517,Z 365.884,A -85,B 0,C 180,E1 25013.824,E2 25013.824} C_VEL
LIN {X 0,Y 520.559,Z 365.884,A -85,B 0,C 180,E1 25010.492,E2 25010.492} C_VEL
LIN {X 0,Y 520.543,Z 365.892,A -85,B 0,C 180,E1 25007.238,E2 25007.238} C_VEL
LIN {X 0,Y 520.529,Z 365.891,A -85,B 0,C 180,E1 25003.806,E2 25003.806} C_VEL
LIN {X 0,Y 520.586,Z 365.885,A -85,B 0,C 180,E1 25000.476,E2 25000.476} C_VEL
LIN {X 0,Y 520.536,Z 365.89,A -85,B 0,C 180,E1 24997.169,E2 24997.169} C_VEL
LIN {X 0,Y 520.543,Z 365.886,A -85,B 0,C 180,E1 24993.659,E2 24993.659} C_VEL
LIN {X 0,Y 520.59,Z 365.885,A -85,B 0,C 180,E1 24990.296,E2 24990.296} C_VEL
LIN {X 0,Y 520.542,Z 365.892,A -85,B 0,C 180,E1 24986.94,E2 24986.94} C_VEL
LIN {X 0,Y 520.556,Z 365.887,A -85,B 0,C 180,E1 24983.456,E2 24983.456} C_VEL
LIN {X 0,Y 520.587,Z 365.872,A -85,B 0,C 180,E1 24980.096,E2 24980.096} C_VEL
LIN {X 0,Y 520.587,Z 365.885,A -85,B 0,C 180,E1 24977.803,E2 24977.803} C_VEL
LIN {X 0,Y 519.587,Z 366.006,A -85,B 0,C 180,E1 24976.955,E2 24976.955} C_VEL
LIN {X 0,Y 513.173,Z 366.8,A -85,B 0,C 180,E1 24974.574,E2 24974.574} C_VEL
LIN {X 0,Y 512.647,Z 366.875,A -85,B 0,C 180,E1 24973.953,E2 24973.953} C_VEL
LIN {X 0,Y 512.612,Z 366.862,A -85,B 0,C 180,E1 24970.474,E2 24970.474} C_VEL
LIN {X 0,Y 512.631,Z 366.857,A -85,B 0,C 180,E1 24967.058,E2 24967.058} C_VEL
LIN {X 0,Y 512.68,Z 367.114,A -85,B 0,C 180,E1 24965.61,E2 24965.61} C_VEL
LIN {X 0,Y 519.518,Z 384.901,A -85,B 0,C 180,E1 24963.129,E2 24963.129} C_VEL
LIN {X 0,Y 522.408,Z 390.43,A -85,B 0,C 180,E1 24962.76,E2 24962.76} C_VEL
LIN {X 0,Y 523.764,Z 393.681,A -85,B 0,C 180,E1 24962.6,E2 24962.6} C_VEL
LIN {X 0,Y 525.183,Z 401.917,A -85,B 0,C 180,E1 24962.352,E2 24962.352} C_VEL
LIN {X 0,Y 522.375,Z 630.519,A -85,B 0,C 180,E1 24958.896,E2 24958.896} C_VEL
LIN {X 0,Y 521.903,Z 652.357,A -85,B 0,C 180,E1 24958.484,E2 24958.484} C_VEL
LIN {X 0,Y 521.184,Z 672.809,A -85,B 0,C 180,E1 24957.888,E2 24957.888} C_VEL
LIN {X 0,Y 520.311,Z 691.168,A -85,B 0,C 180,E1 24957.161,E2 24957.161} C_VEL
LIN {X 0,Y 519.276,Z 709.238,A -85,B 0,C 180,E1 24956.241,E2 24956.241} C_VEL
LIN {X 0,Y 517.903,Z 731.64,A -85,B 0,C 180,E1 24954.825,E2 24954.825} C_VEL
LIN {X 0,Y 516.838,Z 749.289,A -85,B 0,C 180,E1 24953.483,E2 24953.483} C_VEL
LIN {X 0,Y 515.757,Z 766.34,A -85,B 0,C 180,E1 24951.929,E2 24951.929} C_VEL
LIN {X 0,Y 514.81,Z 781.715,A -85,B 0,C 180,E1 24950.268,E2 24950.268} C_VEL
LIN {X 0,Y 513.985,Z 795.788,A -85,B 0,C 180,E1 24948.484,E2 24948.484} C_VEL
LIN {X 0,Y 513.284,Z 808.926,A -85,B 0,C 180,E1 24946.521,E2 24946.521} C_VEL
LIN {X 0,Y 512.747,Z 820.556,A -85,B 0,C 180,E1 24944.452,E2 24944.452} C_VEL
LIN {X 0,Y 512.382,Z 830.209,A -85,B 0,C 180,E1 24942.394,E2 24942.394} C_VEL
LIN {X 0,Y 512.129,Z 838.431,A -85,B 0,C 180,E1 24940.232,E2 24940.232} C_VEL
LIN {X 0,Y 512.003,Z 844.916,A -85,B 0,C 180,E1 24938.072,E2 24938.072} C_VEL
LIN {X 0,Y 511.934,Z 850.179,A -85,B 0,C 180,E1 24935.716,E2 24935.716} C_VEL
LIN {X 0,Y 511.905,Z 853.509,A -85,B 0,C 180,E1 24933.471,E2 24933.471} C_VEL
LIN {X 0,Y 511.903,Z 855.244,A -85,B 0,C 180,E1 24931.231,E2 24931.231} C_VEL
LIN {X 0,Y 511.911,Z 855.313,A -85,B 0,C 180,E1 24928.992,E2 24928.992} C_VEL
LIN {X 0,Y 511.905,Z 853.826,A -85,B 0,C 180,E1 24926.753,E2 24926.753} C_VEL
LIN {X 0,Y 511.919,Z 850.758,A -85,B 0,C 180,E1 24924.508,E2 24924.508} C_VEL
LIN {X 0,Y 511.986,Z 846.039,A -85,B 0,C 180,E1 24922.256,E2 24922.256} C_VEL
LIN {X 0,Y 512.108,Z 839.494,A -85,B 0,C 180,E1 24919.994,E2 24919.994} C_VEL
LIN {X 0,Y 512.326,Z 831.484,A -85,B 0,C 180,E1 24917.833,E2 24917.833} C_VEL
LIN {X 0,Y 512.699,Z 821.567,A -85,B 0,C 180,E1 24915.661,E2 24915.661} C_VEL
LIN {X 0,Y 513.22,Z 810.159,A -85,B 0,C 180,E1 24913.592,E2 24913.592} C_VEL
LIN {X 0,Y 513.868,Z 797.932,A -85,B 0,C 180,E1 24911.719,E2 24911.719} C_VEL
LIN {X 0,Y 514.72,Z 783.379,A -85,B 0,C 180,E1 24909.832,E2 24909.832} C_VEL
LIN {X 0,Y 515.701,Z 767.453,A -85,B 0,C 180,E1 24908.09,E2 24908.09} C_VEL
LIN {X 0,Y 516.771,Z 750.278,A -85,B 0,C 180,E1 24906.513,E2 24906.513} C_VEL
LIN {X 0,Y 517.825,Z 732.744,A -85,B 0,C 180,E1 24905.165,E2 24905.165} C_VEL
LIN {X 0,Y 519.228,Z 710.051,A -85,B 0,C 180,E1 24903.713,E2 24903.713} C_VEL
LIN {X 0,Y 520.265,Z 691.882,A -85,B 0,C 180,E1 24902.783,E2 24902.783} C_VEL
LIN {X 0,Y 521.184,Z 672.811,A -85,B 0,C 180,E1 24902.022,E2 24902.022} C_VEL
LIN {X 0,Y 521.904,Z 652.51,A -85,B 0,C 180,E1 24901.429,E2 24901.429} C_VEL
LIN {X 0,Y 522.379,Z 630.473,A -85,B 0,C 180,E1 24901.014,E2 24901.014} C_VEL
LIN {X 0,Y 525.188,Z 402.907,A -85,B 0,C 180,E1 24897.57,E2 24897.57} C_VEL
LIN {X 0,Y 524.848,Z 399.054,A -85,B 0,C 180,E1 24897.482,E2 24897.482} C_VEL
LIN {X 0,Y 523.179,Z 391.897,A -85,B 0,C 180,E1 24897.235,E2 24897.235} C_VEL
LIN {X 0,Y 519.648,Z 385.24,A -85,B 0,C 180,E1 24896.824,E2 24896.824} C_VEL
LIN {X 0,Y 513.471,Z 369.548,A -85,B 0,C 180,E1 24894.67,E2 24894.67} C_VEL
LIN {X 0,Y 512.663,Z 367.009,A -85,B 0,C 180,E1 24894.263,E2 24894.263} C_VEL
LIN {X 0,Y 512.646,Z 366.879,A -85,B 0,C 180,E1 24890.742,E2 24890.742} C_VEL
LIN {X 0,Y 512.615,Z 366.88,A -85,B 0,C 180,E1 24887.257,E2 24887.257} C_VEL
LIN {X 0,Y 512.641,Z 366.857,A -85,B 0,C 180,E1 24883.815,E2 24883.815} C_VEL
LIN {X 0,Y 512.65,Z 366.871,A -85,B 0,C 180,E1 24880.313,E2 24880.313} C_VEL
LIN {X 0,Y 512.609,Z 366.877,A -85,B 0,C 180,E1 24876.904,E2 24876.904} C_VEL
LIN {X 0,Y 512.631,Z 366.878,A -85,B 0,C 180,E1 24873.414,E2 24873.414} C_VEL
LIN {X 0,Y 512.655,Z 366.869,A -85,B 0,C 180,E1 24869.953,E2 24869.953} C_VEL
LIN {X 0,Y 512.601,Z 366.875,A -85,B 0,C 180,E1 24866.531,E2 24866.531} C_VEL
LIN {X 0,Y 512.62,Z 366.874,A -85,B 0,C 180,E1 24863.082,E2 24863.082} C_VEL
LIN {X 0,Y 512.637,Z 366.876,A -85,B 0,C 180,E1 24859.72,E2 24859.72} C_VEL
LIN {X 0,Y 512.591,Z 366.879,A -85,B 0,C 180,E1 24856.313,E2 24856.313} C_VEL
LIN {X 0,Y 512.627,Z 366.883,A -85,B 0,C 180,E1 24852.962,E2 24852.962} C_VEL
LIN {X 0,Y 512.608,Z 366.873,A -85,B 0,C 180,E1 24849.657,E2 24849.657} C_VEL
LIN {X 0,Y 512.585,Z 366.872,A -85,B 0,C 180,E1 24846.271,E2 24846.271} C_VEL
LIN {X 0,Y 512.638,Z 366.877,A -85,B 0,C 180,E1 24842.907,E2 24842.907} C_VEL
LIN {X 0,Y 512.587,Z 366.881,A -85,B 0,C 180,E1 24839.553,E2 24839.553} C_VEL
LIN {X 0,Y 512.581,Z 366.882,A -85,B 0,C 180,E1 24836.086,E2 24836.086} C_VEL
LIN {X 0,Y 512.646,Z 366.872,A -85,B 0,C 180,E1 24832.717,E2 24832.717} C_VEL
LIN {X 0,Y 512.568,Z 366.88,A -85,B 0,C 180,E1 24829.434,E2 24829.434} C_VEL
LIN {X 0,Y 512.583,Z 366.881,A -85,B 0,C 180,E1 24826.003,E2 24826.003} C_VEL
LIN {X 0,Y 512.598,Z 366.884,A -85,B 0,C 180,E1 24822.754,E2 24822.754} C_VEL
LIN {X 0,Y 512.564,Z 366.885,A -85,B 0,C 180,E1 24819.431,E2 24819.431} C_VEL
LIN {X 0,Y 512.627,Z 366.853,A -85,B 0,C 180,E1 24816.16,E2 24816.16} C_VEL
LIN {X 0,Y 512.579,Z 366.885,A -85,B 0,C 180,E1 24812.799,E2 24812.799} C_VEL
LIN {X 0,Y 512.574,Z 366.862,A -85,B 0,C 180,E1 24809.265,E2 24809.265} C_VEL
LIN {X 0,Y 512.637,Z 366.872,A -85,B 0,C 180,E1 24805.96,E2 24805.96} C_VEL
LIN {X 0,Y 512.582,Z 366.882,A -85,B 0,C 180,E1 24802.653,E2 24802.653} C_VEL
LIN {X 0,Y 512.595,Z 366.866,A -85,B 0,C 180,E1 24799.179,E2 24799.179} C_VEL
LIN {X 0,Y 512.631,Z 366.856,A -85,B 0,C 180,E1 24795.865,E2 24795.865} C_VEL
LIN {X 0,Y 512.638,Z 367.167,A -85,B 0,C 180,E1 24794.993,E2 24794.993} C_VEL
LIN {X 0,Y 513.901,Z 370.379,A -85,B 0,C 180,E1 24794.595,E2 24794.595} C_VEL
LIN {X 0,Y 521.726,Z 386.804,A -85,B 0,C 180,E1 24792.778,E2 24792.778} C_VEL
LIN {X 0,Y 527.85,Z 400.047,A -85,B 0,C 180,E1 24791.401,E2 24791.401} C_VEL
LIN {X 0,Y 526.088,Z 453.503,A -85,B 0,C 180,E1 24788.177,E2 24788.177} C_VEL
LIN {X 0,Y 528.635,Z 472.225,A -85,B 0,C 180,E1 24787.662,E2 24787.662} C_VEL
LIN {X 0,Y 526.586,Z 644.464,A -85,B 0,C 180,E1 24785.025,E2 24785.025} C_VEL
LIN {X 0,Y 525.045,Z 761.901,A -85,B 0,C 180,E1 24783.204,E2 24783.204} C_VEL
LIN {X 0,Y 524.289,Z 783.349,A -85,B 0,C 180,E1 24782.676,E2 24782.676} C_VEL
LIN {X 0,Y 523.338,Z 805.539,A -85,B 0,C 180,E1 24781.917,E2 24781.917} C_VEL
LIN {X 0,Y 522.317,Z 825.214,A -85,B 0,C 180,E1 24781.054,E2 24781.054} C_VEL
LIN {X 0,Y 521.071,Z 844.79,A -85,B 0,C 180,E1 24779.988,E2 24779.988} C_VEL
LIN {X 0,Y 519.708,Z 865.536,A -85,B 0,C 180,E1 24778.621,E2 24778.621} C_VEL
LIN {X 0,Y 518.438,Z 883.782,A -85,B 0,C 180,E1 24777.196,E2 24777.196} C_VEL
LIN {X 0,Y 517.112,Z 901.725,A -85,B 0,C 180,E1 24775.54,E2 24775.54} C_VEL
LIN {X 0,Y 515.899,Z 918.687,A -85,B 0,C 180,E1 24773.711,E2 24773.711} C_VEL
LIN {X 0,Y 514.845,Z 934.188,A -85,B 0,C 180,E1 24771.771,E2 24771.771} C_VEL
LIN {X 0,Y 513.936,Z 948.641,A -85,B 0,C 180,E1 24769.666,E2 24769.666} C_VEL
LIN {X 0,Y 513.212,Z 961.464,A -85,B 0,C 180,E1 24767.458,E2 24767.458} C_VEL
LIN {X 0,Y 512.674,Z 972.82,A -85,B 0,C 180,E1 24765.148,E2 24765.148} C_VEL
LIN {X 0,Y 512.323,Z 982.26,A -85,B 0,C 180,E1 24762.854,E2 24762.854} C_VEL
LIN {X 0,Y 512.109,Z 989.884,A -85,B 0,C 180,E1 24760.575,E2 24760.575} C_VEL
LIN {X 0,Y 511.989,Z 996.146,A -85,B 0,C 180,E1 24758.196,E2 24758.196} C_VEL
LIN {X 0,Y 511.933,Z 1000.823,A -85,B 0,C 180,E1 24755.829,E2 24755.829} C_VEL
LIN {X 0,Y 511.913,Z 1003.786,A -85,B 0,C 180,E1 24753.471,E2 24753.471} C_VEL
LIN {X 0,Y 511.907,Z 1005.305,A -85,B 0,C 180,E1 24751.008,E2 24751.008} C_VEL
LIN {X 0,Y 511.906,Z 1005.237,A -85,B 0,C 180,E1 24748.657,E2 24748.657} C_VEL
LIN {X 0,Y 511.91,Z 1003.56,A -85,B 0,C 180,E1 24746.305,E2 24746.305} C_VEL
LIN {X 0,Y 511.937,Z 1000.428,A -85,B 0,C 180,E1 24743.947,E2 24743.947} C_VEL
LIN {X 0,Y 511.996,Z 995.639,A -85,B 0,C 180,E1 24741.579,E2 24741.579} C_VEL
LIN {X 0,Y 512.124,Z 988.95,A -85,B 0,C 180,E1 24739.125,E2 24739.125} C_VEL
LIN {X 0,Y 512.366,Z 980.979,A -85,B 0,C 180,E1 24736.804,E2 24736.804} C_VEL
LIN {X 0,Y 512.746,Z 971.269,A -85,B 0,C 180,E1 24734.507,E2 24734.507} C_VEL
LIN {X 0,Y 513.286,Z 960.019,A -85,B 0,C 180,E1 24732.278,E2 24732.278} C_VEL
LIN {X 0,Y 514.02,Z 947.113,A -85,B 0,C 180,E1 24730.101,E2 24730.101} C_VEL
LIN {X 0,Y 514.961,Z 932.493,A -85,B 0,C 180,E1 24727.995,E2 24727.995} C_VEL
LIN {X 0,Y 516.044,Z 916.668,A -85,B 0,C 180,E1 24726.054,E2 24726.054} C_VEL
LIN {X 0,Y 517.264,Z 899.651,A -85,B 0,C 180,E1 24724.258,E2 24724.258} C_VEL
LIN {X 0,Y 518.568,Z 881.626,A -85,B 0,C 180,E1 24722.626,E2 24722.626} C_VEL
LIN {X 0,Y 519.896,Z 863.119,A -85,B 0,C 180,E1 24721.203,E2 24721.203} C_VEL
LIN {X 0,Y 521.131,Z 843.803,A -85,B 0,C 180,E1 24719.953,E2 24719.953} C_VEL
LIN {X 0,Y 522.426,Z 823.108,A -85,B 0,C 180,E1 24718.847,E2 24718.847} C_VEL
LIN {X 0,Y 523.431,Z 803.696,A -85,B 0,C 180,E1 24718.008,E2 24718.008} C_VEL
LIN {X 0,Y 524.333,Z 782.353,A -85,B 0,C 180,E1 24717.295,E2 24717.295} C_VEL
LIN {X 0,Y 525.061,Z 760.884,A -85,B 0,C 180,E1 24716.778,E2 24716.778} C_VEL
LIN {X 0,Y 527.845,Z 546.946,A -85,B 0,C 180,E1 24713.471,E2 24713.471} C_VEL
LIN {X 0,Y 528.475,Z 469.69,A -85,B 0,C 180,E1 24712.284,E2 24712.284} C_VEL
LIN {X 0,Y 526.088,Z 453.519,A -85,B 0,C 180,E1 24711.824,E2 24711.824} C_VEL
LIN {X 0,Y 527.863,Z 399.688,A -85,B 0,C 180,E1 24708.577,E2 24708.577} C_VEL
LIN {X 0,Y 514.432,Z 371.086,A -85,B 0,C 180,E1 24705.504,E2 24705.504} C_VEL
LIN {X 0,Y 512.744,Z 367.719,A -85,B 0,C 180,E1 24705.104,E2 24705.104} C_VEL
LIN {X 0,Y 512.608,Z 366.91,A -85,B 0,C 180,E1 24704.918,E2 24704.918} C_VEL
LIN {X 0,Y 512.587,Z 366.879,A -85,B 0,C 180,E1 24701.5,E2 24701.5} C_VEL
LIN {X 0,Y 512.647,Z 366.878,A -85,B 0,C 180,E1 24698.19,E2 24698.19} C_VEL
LIN {X 0,Y 512.581,Z 366.87,A -85,B 0,C 180,E1 24694.802,E2 24694.802} C_VEL
LIN {X 0,Y 512.579,Z 366.867,A -85,B 0,C 180,E1 24691.256,E2 24691.256} C_VEL
LIN {X 0,Y 512.643,Z 366.876,A -85,B 0,C 180,E1 24687.94,E2 24687.94} C_VEL
LIN {X 0,Y 512.568,Z 366.859,A -85,B 0,C 180,E1 24684.55,E2 24684.55} C_VEL
LIN {X 0,Y 512.576,Z 366.885,A -85,B 0,C 180,E1 24681.034,E2 24681.034} C_VEL
LIN {X 0,Y 512.622,Z 366.879,A -85,B 0,C 180,E1 24677.714,E2 24677.714} C_VEL
LIN {X 0,Y 512.561,Z 366.881,A -85,B 0,C 180,E1 24674.459,E2 24674.459} C_VEL
LIN {X 0,Y 512.608,Z 366.877,A -85,B 0,C 180,E1 24671.134,E2 24671.134} C_VEL
LIN {X 0,Y 512.582,Z 366.882,A -85,B 0,C 180,E1 24667.848,E2 24667.848} C_VEL
LIN {X 0,Y 512.573,Z 366.882,A -85,B 0,C 180,E1 24664.363,E2 24664.363} C_VEL
LIN {X 0,Y 512.638,Z 366.882,A -85,B 0,C 180,E1 24661.006,E2 24661.006} C_VEL
LIN {X 0,Y 512.586,Z 366.874,A -85,B 0,C 180,E1 24657.652,E2 24657.652} C_VEL
LIN {X 0,Y 512.581,Z 366.872,A -85,B 0,C 180,E1 24654.108,E2 24654.108} C_VEL
LIN {X 0,Y 512.645,Z 366.874,A -85,B 0,C 180,E1 24650.797,E2 24650.797} C_VEL
LIN {X 0,Y 512.589,Z 366.881,A -85,B 0,C 180,E1 24647.495,E2 24647.495} C_VEL
LIN {X 0,Y 512.595,Z 366.879,A -85,B 0,C 180,E1 24643.92,E2 24643.92} C_VEL
LIN {X 0,Y 512.643,Z 366.873,A -85,B 0,C 180,E1 24640.636,E2 24640.636} C_VEL
LIN {X 0,Y 512.595,Z 366.878,A -85,B 0,C 180,E1 24637.281,E2 24637.281} C_VEL
LIN {X 0,Y 512.612,Z 366.874,A -85,B 0,C 180,E1 24633.785,E2 24633.785} C_VEL
LIN {X 0,Y 512.646,Z 366.877,A -85,B 0,C 180,E1 24630.432,E2 24630.432} C_VEL
LIN {X 0,Y 512.601,Z 366.881,A -85,B 0,C 180,E1 24626.998,E2 24626.998} C_VEL
LIN {X 0,Y 512.62,Z 366.876,A -85,B 0,C 180,E1 24623.494,E2 24623.494} C_VEL
LIN {X 0,Y 512.647,Z 366.86,A -85,B 0,C 180,E1 24620.033,E2 24620.033} C_VEL
LIN {X 0,Y 512.609,Z 366.868,A -85,B 0,C 180,E1 24616.639,E2 24616.639} C_VEL
LIN {X 0,Y 512.647,Z 366.875,A -85,B 0,C 180,E1 24613.953,E2 24613.953} C_VEL
LIN {X 0,Y 511.654,Z 367.006,A -85,B 0,C 180,E1 24613.092,E2 24613.092} C_VEL
LIN {X 0,Y 505.205,Z 367.784,A -85,B 0,C 180,E1 24610.672,E2 24610.672} C_VEL
LIN {X 0,Y 504.697,Z 367.854,A -85,B 0,C 180,E1 24610.042,E2 24610.042} C_VEL
LIN {X 0,Y 504.673,Z 367.85,A -85,B 0,C 180,E1 24606.603,E2 24606.603} C_VEL
LIN {X 0,Y 504.727,Z 368.182,A -85,B 0,C 180,E1 24606.267,E2 24606.267} C_VEL
LIN {X 0,Y 511.474,Z 385.259,A -85,B 0,C 180,E1 24603.817,E2 24603.817} C_VEL
LIN {X 0,Y 512.908,Z 388.047,A -85,B 0,C 180,E1 24603.579,E2 24603.579} C_VEL
LIN {X 0,Y 517.601,Z 396.873,A -85,B 0,C 180,E1 24603.044,E2 24603.044} C_VEL
LIN {X 0,Y 518.689,Z 403.495,A -85,B 0,C 180,E1 24602.848,E2 24602.848} C_VEL
LIN {X 0,Y 515.704,Z 633.659,A -85,B 0,C 180,E1 24599.345,E2 24599.345} C_VEL
LIN {X 0,Y 515.229,Z 654.449,A -85,B 0,C 180,E1 24598.937,E2 24598.937} C_VEL
LIN {X 0,Y 514.473,Z 674.471,A -85,B 0,C 180,E1 24598.34,E2 24598.34} C_VEL
LIN {X 0,Y 513.552,Z 692.764,A -85,B 0,C 180,E1 24597.602,E2 24597.602} C_VEL
LIN {X 0,Y 512.442,Z 710.975,A -85,B 0,C 180,E1 24596.661,E2 24596.661} C_VEL
LIN {X 0,Y 511.095,Z 729.167,A -85,B 0,C 180,E1 24595.489,E2 24595.489} C_VEL
LIN {X 0,Y 509.767,Z 745.668,A -85,B 0,C 180,E1 24594.198,E2 24594.198} C_VEL
LIN {X 0,Y 508.097,Z 767.731,A -85,B 0,C 180,E1 24592.135,E2 24592.135} C_VEL
LIN {X 0,Y 507.013,Z 783.796,A -85,B 0,C 180,E1 24590.346,E2 24590.346} C_VEL
LIN {X 0,Y 506.078,Z 798.322,A -85,B 0,C 180,E1 24588.426,E2 24588.426} C_VEL
LIN {X 0,Y 505.333,Z 811.026,A -85,B 0,C 180,E1 24586.434,E2 24586.434} C_VEL
LIN {X 0,Y 504.766,Z 822.275,A -85,B 0,C 180,E1 24584.334,E2 24584.334} C_VEL
LIN {X 0,Y 504.361,Z 832.049,A -85,B 0,C 180,E1 24582.129,E2 24582.129} C_VEL
LIN {X 0,Y 504.12,Z 839.933,A -85,B 0,C 180,E1 24579.935,E2 24579.935} C_VEL
LIN {X 0,Y 503.988,Z 846.38,A -85,B 0,C 180,E1 24577.637,E2 24577.637} C_VEL
LIN {X 0,Y 503.92,Z 851.003,A -85,B 0,C 180,E1 24575.35,E2 24575.35} C_VEL
LIN {X 0,Y 503.905,Z 853.963,A -85,B 0,C 180,E1 24573.07,E2 24573.07} C_VEL
LIN {X 0,Y 503.906,Z 855.363,A -85,B 0,C 180,E1 24570.682,E2 24570.682} C_VEL
LIN {X 0,Y 503.9,Z 855.102,A -85,B 0,C 180,E1 24568.408,E2 24568.408} C_VEL
LIN {X 0,Y 503.916,Z 853.255,A -85,B 0,C 180,E1 24566.132,E2 24566.132} C_VEL
LIN {X 0,Y 503.948,Z 849.721,A -85,B 0,C 180,E1 24563.85,E2 24563.85} C_VEL
LIN {X 0,Y 504.026,Z 844.522,A -85,B 0,C 180,E1 24561.559,E2 24561.559} C_VEL
LIN {X 0,Y 504.191,Z 837.533,A -85,B 0,C 180,E1 24559.257,E2 24559.257} C_VEL
LIN {X 0,Y 504.487,Z 829.095,A -85,B 0,C 180,E1 24557.059,E2 24557.059} C_VEL
LIN {X 0,Y 504.945,Z 818.666,A -85,B 0,C 180,E1 24554.849,E2 24554.849} C_VEL
LIN {X 0,Y 505.586,Z 806.641,A -85,B 0,C 180,E1 24552.745,E2 24552.745} C_VEL
LIN {X 0,Y 506.349,Z 793.884,A -85,B 0,C 180,E1 24550.867,E2 24550.867} C_VEL
LIN {X 0,Y 507.304,Z 779.313,A -85,B 0,C 180,E1 24549.041,E2 24549.041} C_VEL
LIN {X 0,Y 508.403,Z 763.177,A -85,B 0,C 180,E1 24547.329,E2 24547.329} C_VEL
LIN {X 0,Y 509.857,Z 744.583,A -85,B 0,C 180,E1 24545.621,E2 24545.621} C_VEL
LIN {X 0,Y 511.248,Z 726.983,A -85,B 0,C 180,E1 24544.27,E2 24544.27} C_VEL
LIN {X 0,Y 512.538,Z 709.297,A -85,B 0,C 180,E1 24543.155,E2 24543.155} C_VEL
LIN {X 0,Y 513.672,Z 690.807,A -85,B 0,C 180,E1 24542.216,E2 24542.216} C_VEL
LIN {X 0,Y 514.614,Z 671.618,A -85,B 0,C 180,E1 24541.47,E2 24541.47} C_VEL
LIN {X 0,Y 515.31,Z 651.487,A -85,B 0,C 180,E1 24540.902,E2 24540.902} C_VEL
LIN {X 0,Y 515.845,Z 623.968,A -85,B 0,C 180,E1 24540.415,E2 24540.415} C_VEL
LIN {X 0,Y 518.686,Z 402.312,A -85,B 0,C 180,E1 24537.042,E2 24537.042} C_VEL
LIN {X 0,Y 517.091,Z 395.529,A -85,B 0,C 180,E1 24536.802,E2 24536.802} C_VEL
LIN {X 0,Y 511.647,Z 385.727,A -85,B 0,C 180,E1 24536.154,E2 24536.154} C_VEL
LIN {X 0,Y 505.511,Z 370.504,A -85,B 0,C 180,E1 24533.996,E2 24533.996} C_VEL
LIN {X 0,Y 504.714,Z 368.077,A -85,B 0,C 180,E1 24533.611,E2 24533.611} C_VEL
LIN {X 0,Y 504.706,Z 367.864,A -85,B 0,C 180,E1 24530.369,E2 24530.369} C_VEL
LIN {X 0,Y 504.685,Z 367.868,A -85,B 0,C 180,E1 24526.887,E2 24526.887} C_VEL
LIN {X 0,Y 504.677,Z 367.852,A -85,B 0,C 180,E1 24523.362,E2 24523.362} C_VEL
LIN {X 0,Y 504.71,Z 367.848,A -85,B 0,C 180,E1 24519.931,E2 24519.931} C_VEL
LIN {X 0,Y 504.687,Z 367.864,A -85,B 0,C 180,E1 24516.46,E2 24516.46} C_VEL
LIN {X 0,Y 504.669,Z 367.87,A -85,B 0,C 180,E1 24513.014,E2 24513.014} C_VEL
LIN {X 0,Y 504.71,Z 367.864,A -85,B 0,C 180,E1 24509.557,E2 24509.557} C_VEL
LIN {X 0,Y 504.686,Z 367.862,A -85,B 0,C 180,E1 24506.092,E2 24506.092} C_VEL
LIN {X 0,Y 504.658,Z 367.865,A -85,B 0,C 180,E1 24502.605,E2 24502.605} C_VEL
LIN {X 0,Y 504.698,Z 367.86,A -85,B 0,C 180,E1 24499.2,E2 24499.2} C_VEL
LIN {X 0,Y 504.683,Z 367.866,A -85,B 0,C 180,E1 24495.749,E2 24495.749} C_VEL
LIN {X 0,Y 504.65,Z 367.87,A -85,B 0,C 180,E1 24492.356,E2 24492.356} C_VEL
LIN {X 0,Y 504.7,Z 367.867,A -85,B 0,C 180,E1 24489.004,E2 24489.004} C_VEL
LIN {X 0,Y 504.654,Z 367.86,A -85,B 0,C 180,E1 24485.686,E2 24485.686} C_VEL
LIN {X 0,Y 504.643,Z 367.863,A -85,B 0,C 180,E1 24482.158,E2 24482.158} C_VEL
LIN {X 0,Y 504.704,Z 367.869,A -85,B 0,C 180,E1 24478.865,E2 24478.865} C_VEL
LIN {X 0,Y 504.643,Z 367.871,A -85,B 0,C 180,E1 24475.455,E2 24475.455} C_VEL
LIN {X 0,Y 504.636,Z 367.871,A -85,B 0,C 180,E1 24471.913,E2 24471.913} C_VEL
LIN {X 0,Y 504.692,Z 367.862,A -85,B 0,C 180,E1 24468.574,E2 24468.574} C_VEL
LIN {X 0,Y 504.627,Z 367.869,A -85,B 0,C 180,E1 24465.309,E2 24465.309} C_VEL
LIN {X 0,Y 504.633,Z 367.868,A -85,B 0,C 180,E1 24461.757,E2 24461.757} C_VEL
LIN {X 0,Y 504.689,Z 367.867,A -85,B 0,C 180,E1 24458.378,E2 24458.378} C_VEL
LIN {X 0,Y 504.629,Z 367.851,A -85,B 0,C 180,E1 24455.037,E2 24455.037} C_VEL
LIN {X 0,Y 504.651,Z 367.867,A -85,B 0,C 180,E1 24451.595,E2 24451.595} C_VEL
LIN {X 0,Y 504.67,Z 367.855,A -85,B 0,C 180,E1 24448.331,E2 24448.331} C_VEL
LIN {X 0,Y 504.637,Z 367.854,A -85,B 0,C 180,E1 24444.907,E2 24444.907} C_VEL
LIN {X 0,Y 504.678,Z 367.867,A -85,B 0,C 180,E1 24441.49,E2 24441.49} C_VEL
LIN {X 0,Y 504.673,Z 367.87,A -85,B 0,C 180,E1 24438.147,E2 24438.147} C_VEL
LIN {X 0,Y 504.73,Z 368.038,A -85,B 0,C 180,E1 24435.725,E2 24435.725} C_VEL
LIN {X 0,Y 505.271,Z 369.989,A -85,B 0,C 180,E1 24435.453,E2 24435.453} C_VEL
LIN {X 0,Y 512.293,Z 384.509,A -85,B 0,C 180,E1 24433.769,E2 24433.769} C_VEL
LIN {X 0,Y 521.088,Z 403.385,A -85,B 0,C 180,E1 24431.741,E2 24431.741} C_VEL
LIN {X 0,Y 519.29,Z 453.651,A -85,B 0,C 180,E1 24428.684,E2 24428.684} C_VEL
LIN {X 0,Y 522.006,Z 473.524,A -85,B 0,C 180,E1 24428.137,E2 24428.137} C_VEL
LIN {X 0,Y 519.344,Z 695.736,A -85,B 0,C 180,E1 24424.738,E2 24424.738} C_VEL
LIN {X 0,Y 518.333,Z 762.694,A -85,B 0,C 180,E1 24423.675,E2 24423.675} C_VEL
LIN {X 0,Y 517.511,Z 783.999,A -85,B 0,C 180,E1 24423.138,E2 24423.138} C_VEL
LIN {X 0,Y 516.456,Z 806.276,A -85,B 0,C 180,E1 24422.361,E2 24422.361} C_VEL
LIN {X 0,Y 515.313,Z 826.433,A -85,B 0,C 180,E1 24421.459,E2 24421.459} C_VEL
LIN {X 0,Y 513.901,Z 846.796,A -85,B 0,C 180,E1 24420.321,E2 24420.321} C_VEL
LIN {X 0,Y 512.477,Z 866.344,A -85,B 0,C 180,E1 24418.999,E2 24418.999} C_VEL
LIN {X 0,Y 511.083,Z 884.452,A -85,B 0,C 180,E1 24417.558,E2 24417.558} C_VEL
LIN {X 0,Y 509.652,Z 902.291,A -85,B 0,C 180,E1 24415.883,E2 24415.883} C_VEL
LIN {X 0,Y 508.389,Z 918.223,A -85,B 0,C 180,E1 24414.14,E2 24414.14} C_VEL
LIN {X 0,Y 507.244,Z 933.338,A -85,B 0,C 180,E1 24412.237,E2 24412.237} C_VEL
LIN {X 0,Y 506.225,Z 947.877,A -85,B 0,C 180,E1 24410.099,E2 24410.099} C_VEL
LIN {X 0,Y 505.424,Z 960.529,A -85,B 0,C 180,E1 24407.911,E2 24407.911} C_VEL
LIN {X 0,Y 504.796,Z 972.304,A -85,B 0,C 180,E1 24405.508,E2 24405.508} C_VEL
LIN {X 0,Y 504.392,Z 981.853,A -85,B 0,C 180,E1 24403.176,E2 24403.176} C_VEL
LIN {X 0,Y 504.138,Z 989.531,A -85,B 0,C 180,E1 24400.86,E2 24400.86} C_VEL
LIN {X 0,Y 503.999,Z 996.146,A -85,B 0,C 180,E1 24398.326,E2 24398.326} C_VEL
LIN {X 0,Y 503.934,Z 1000.823,A -85,B 0,C 180,E1 24395.922,E2 24395.922} C_VEL
LIN {X 0,Y 503.914,Z 1003.787,A -85,B 0,C 180,E1 24393.527,E2 24393.527} C_VEL
LIN {X 0,Y 503.907,Z 1005.305,A -85,B 0,C 180,E1 24391.024,E2 24391.024} C_VEL
LIN {X 0,Y 503.908,Z 1005.259,A -85,B 0,C 180,E1 24388.75,E2 24388.75} C_VEL
LIN {X 0,Y 503.911,Z 1003.673,A -85,B 0,C 180,E1 24386.36,E2 24386.36} C_VEL
LIN {X 0,Y 503.938,Z 1000.634,A -85,B 0,C 180,E1 24383.965,E2 24383.965} C_VEL
LIN {X 0,Y 504.002,Z 995.893,A -85,B 0,C 180,E1 24381.559,E2 24381.559} C_VEL
LIN {X 0,Y 504.144,Z 989.179,A -85,B 0,C 180,E1 24379.026,E2 24379.026} C_VEL
LIN {X 0,Y 504.408,Z 981.434,A -85,B 0,C 180,E1 24376.708,E2 24376.708} C_VEL
LIN {X 0,Y 504.823,Z 971.789,A -85,B 0,C 180,E1 24374.376,E2 24374.376} C_VEL
LIN {X 0,Y 505.443,Z 960.198,A -85,B 0,C 180,E1 24372.028,E2 24372.028} C_VEL
LIN {X 0,Y 506.225,Z 947.882,A -85,B 0,C 180,E1 24369.902,E2 24369.902} C_VEL
LIN {X 0,Y 507.244,Z 933.344,A -85,B 0,C 180,E1 24367.764,E2 24367.764} C_VEL
LIN {X 0,Y 508.391,Z 918.187,A -85,B 0,C 180,E1 24365.856,E2 24365.856} C_VEL
LIN {X 0,Y 509.744,Z 901.124,A -85,B 0,C 180,E1 24364.002,E2 24364.002} C_VEL
LIN {X 0,Y 511.137,Z 883.792,A -85,B 0,C 180,E1 24362.383,E2 24362.383} C_VEL
LIN {X 0,Y 512.575,Z 865.159,A -85,B 0,C 180,E1 24360.914,E2 24360.914} C_VEL
LIN {X 0,Y 514.028,Z 844.804,A -85,B 0,C 180,E1 24359.559,E2 24359.559} C_VEL
LIN {X 0,Y 515.389,Z 825.236,A -85,B 0,C 180,E1 24358.482,E2 24358.482} C_VEL
LIN {X 0,Y 516.534,Z 804.829,A -85,B 0,C 180,E1 24357.579,E2 24357.579} C_VEL
LIN {X 0,Y 517.56,Z 782.912,A -85,B 0,C 180,E1 24356.83,E2 24356.83} C_VEL
LIN {X 0,Y 518.355,Z 761.634,A -85,B 0,C 180,E1 24356.305,E2 24356.305} C_VEL
LIN {X 0,Y 520,Z 644.767,A -85,B 0,C 180,E1 24354.478,E2 24354.478} C_VEL
LIN {X 0,Y 521.939,Z 471.612,A -85,B 0,C 180,E1 24351.826,E2 24351.826} C_VEL
LIN {X 0,Y 519.239,Z 452.441,A -85,B 0,C 180,E1 24351.262,E2 24351.262} C_VEL
LIN {X 0,Y 521.083,Z 403.146,A -85,B 0,C 180,E1 24348.243,E2 24348.243} C_VEL
LIN {X 0,Y 508.229,Z 375.85,A -85,B 0,C 180,E1 24345.251,E2 24345.251} C_VEL
LIN {X 0,Y 504.788,Z 368.37,A -85,B 0,C 180,E1 24344.359,E2 24344.359} C_VEL
LIN {X 0,Y 504.685,Z 367.844,A -85,B 0,C 180,E1 24344.057,E2 24344.057} C_VEL
LIN {X 0,Y 504.667,Z 367.85,A -85,B 0,C 180,E1 24340.679,E2 24340.679} C_VEL
LIN {X 0,Y 504.641,Z 367.87,A -85,B 0,C 180,E1 24337.212,E2 24337.212} C_VEL
LIN {X 0,Y 504.688,Z 367.865,A -85,B 0,C 180,E1 24333.828,E2 24333.828} C_VEL
LIN {X 0,Y 504.65,Z 367.846,A -85,B 0,C 180,E1 24330.478,E2 24330.478} C_VEL
LIN {X 0,Y 504.64,Z 367.872,A -85,B 0,C 180,E1 24327.11,E2 24327.11} C_VEL
LIN {X 0,Y 504.693,Z 367.839,A -85,B 0,C 180,E1 24323.713,E2 24323.713} C_VEL
LIN {X 0,Y 504.632,Z 367.873,A -85,B 0,C 180,E1 24320.409,E2 24320.409} C_VEL
LIN {X 0,Y 504.628,Z 367.873,A -85,B 0,C 180,E1 24316.815,E2 24316.815} C_VEL
LIN {X 0,Y 504.692,Z 367.872,A -85,B 0,C 180,E1 24313.436,E2 24313.436} C_VEL
LIN {X 0,Y 504.635,Z 367.869,A -85,B 0,C 180,E1 24310.041,E2 24310.041} C_VEL
LIN {X 0,Y 504.633,Z 367.868,A -85,B 0,C 180,E1 24306.484,E2 24306.484} C_VEL
LIN {X 0,Y 504.693,Z 367.861,A -85,B 0,C 180,E1 24303.18,E2 24303.18} C_VEL
LIN {X 0,Y 504.637,Z 367.872,A -85,B 0,C 180,E1 24299.886,E2 24299.886} C_VEL
LIN {X 0,Y 504.651,Z 367.87,A -85,B 0,C 180,E1 24296.365,E2 24296.365} C_VEL
LIN {X 0,Y 504.707,Z 367.861,A -85,B 0,C 180,E1 24292.935,E2 24292.935} C_VEL
LIN {X 0,Y 504.65,Z 367.863,A -85,B 0,C 180,E1 24289.497,E2 24289.497} C_VEL
LIN {X 0,Y 504.65,Z 367.864,A -85,B 0,C 180,E1 24285.895,E2 24285.895} C_VEL
LIN {X 0,Y 504.708,Z 367.867,A -85,B 0,C 180,E1 24282.594,E2 24282.594} C_VEL
LIN {X 0,Y 504.658,Z 367.869,A -85,B 0,C 180,E1 24279.228,E2 24279.228} C_VEL
LIN {X 0,Y 504.661,Z 367.867,A -85,B 0,C 180,E1 24275.663,E2 24275.663} C_VEL
LIN {X 0,Y 504.714,Z 367.863,A -85,B 0,C 180,E1 24272.254,E2 24272.254} C_VEL
LIN {X 0,Y 504.667,Z 367.863,A -85,B 0,C 180,E1 24268.848,E2 24268.848} C_VEL
LIN {X 0,Y 504.667,Z 367.866,A -85,B 0,C 180,E1 24265.297,E2 24265.297} C_VEL
LIN {X 0,Y 504.707,Z 367.837,A -85,B 0,C 180,E1 24261.85,E2 24261.85} C_VEL
LIN {X 0,Y 504.694,Z 367.872,A -85,B 0,C 180,E1 24258.314,E2 24258.314} C_VEL
LIN {X 0,Y 504.669,Z 367.854,A -85,B 0,C 180,E1 24254.824,E2 24254.824} C_VEL
LIN {X 0,Y 504.705,Z 367.842,A -85,B 0,C 180,E1 24251.338,E2 24251.338} C_VEL
LIN {X 0,Y 504.697,Z 367.854,A -85,B 0,C 180,E1 24250.042,E2 24250.042} C_VEL
LIN {X 0,Y 503.716,Z 367.991,A -85,B 0,C 180,E1 24249.46,E2 24249.46} C_VEL
LIN {X 0,Y 497.315,Z 368.768,A -85,B 0,C 180,E1 24247.88,E2 24247.88} C_VEL
LIN {X 0,Y 496.766,Z 368.831,A -85,B 0,C 180,E1 24247.452,E2 24247.452} C_VEL
LIN {X 0,Y 496.784,Z 369.087,A -85,B 0,C 180,E1 24246.993,E2 24246.993} C_VEL
LIN {X 0,Y 503.291,Z 385.416,A -85,B 0,C 180,E1 24244.567,E2 24244.567} C_VEL
LIN {X 0,Y 504.455,Z 387.902,A -85,B 0,C 180,E1 24244.307,E2 24244.307} C_VEL
LIN {X 0,Y 511.506,Z 400.233,A -85,B 0,C 180,E1 24243.494,E2 24243.494} C_VEL
LIN {X 0,Y 512.217,Z 405.278,A -85,B 0,C 180,E1 24243.351,E2 24243.351} C_VEL
LIN {X 0,Y 509.052,Z 637.571,A -85,B 0,C 180,E1 24239.793,E2 24239.793} C_VEL
LIN {X 0,Y 508.56,Z 658.116,A -85,B 0,C 180,E1 24239.364,E2 24239.364} C_VEL
LIN {X 0,Y 507.724,Z 677.609,A -85,B 0,C 180,E1 24238.751,E2 24238.751} C_VEL
LIN {X 0,Y 506.683,Z 696.622,A -85,B 0,C 180,E1 24237.944,E2 24237.944} C_VEL
LIN {X 0,Y 505.493,Z 714.325,A -85,B 0,C 180,E1 24236.994,E2 24236.994} C_VEL
LIN {X 0,Y 504.092,Z 732.232,A -85,B 0,C 180,E1 24235.806,E2 24235.806} C_VEL
LIN {X 0,Y 502.6,Z 749.093,A -85,B 0,C 180,E1 24234.44,E2 24234.44} C_VEL
LIN {X 0,Y 501.13,Z 765.052,A -85,B 0,C 180,E1 24232.893,E2 24232.893} C_VEL
LIN {X 0,Y 499.736,Z 779.849,A -85,B 0,C 180,E1 24231.194,E2 24231.194} C_VEL
LIN {X 0,Y 498.372,Z 797.483,A -85,B 0,C 180,E1 24228.842,E2 24228.842} C_VEL
LIN {X 0,Y 497.539,Z 810.33,A -85,B 0,C 180,E1 24226.819,E2 24226.819} C_VEL
LIN {X 0,Y 496.897,Z 821.706,A -85,B 0,C 180,E1 24224.685,E2 24224.685} C_VEL
LIN {X 0,Y 496.441,Z 831.594,A -85,B 0,C 180,E1 24222.443,E2 24222.443} C_VEL
LIN {X 0,Y 496.156,Z 839.582,A -85,B 0,C 180,E1 24220.213,E2 24220.213} C_VEL
LIN {X 0,Y 496.008,Z 846.1,A -85,B 0,C 180,E1 24217.877,E2 24217.877} C_VEL
LIN {X 0,Y 495.929,Z 850.799,A -85,B 0,C 180,E1 24215.552,E2 24215.552} C_VEL
LIN {X 0,Y 495.903,Z 853.85,A -85,B 0,C 180,E1 24213.236,E2 24213.236} C_VEL
LIN {X 0,Y 495.911,Z 855.318,A -85,B 0,C 180,E1 24210.924,E2 24210.924} C_VEL
LIN {X 0,Y 495.9,Z 855.233,A -85,B 0,C 180,E1 24208.613,E2 24208.613} C_VEL
LIN {X 0,Y 495.91,Z 853.481,A -85,B 0,C 180,E1 24206.301,E2 24206.301} C_VEL
LIN {X 0,Y 495.947,Z 850.133,A -85,B 0,C 180,E1 24203.983,E2 24203.983} C_VEL
LIN {X 0,Y 496.027,Z 845.127,A -85,B 0,C 180,E1 24201.655,E2 24201.655} C_VEL
LIN {X 0,Y 496.189,Z 838.747,A -85,B 0,C 180,E1 24199.434,E2 24199.434} C_VEL
LIN {X 0,Y 496.517,Z 830.097,A -85,B 0,C 180,E1 24197.085,E2 24197.085} C_VEL
LIN {X 0,Y 496.998,Z 819.834,A -85,B 0,C 180,E1 24194.84,E2 24194.84} C_VEL
LIN {X 0,Y 497.637,Z 808.744,A -85,B 0,C 180,E1 24192.823,E2 24192.823} C_VEL
LIN {X 0,Y 498.499,Z 795.571,A -85,B 0,C 180,E1 24190.797,E2 24190.797} C_VEL
LIN {X 0,Y 500.11,Z 775.964,A -85,B 0,C 180,E1 24188.233,E2 24188.233} C_VEL
LIN {X 0,Y 501.6,Z 760.159,A -85,B 0,C 180,E1 24186.507,E2 24186.507} C_VEL
LIN {X 0,Y 503.005,Z 744.524,A -85,B 0,C 180,E1 24185.079,E2 24185.079} C_VEL
LIN {X 0,Y 504.449,Z 727.473,A -85,B 0,C 180,E1 24183.771,E2 24183.771} C_VEL
LIN {X 0,Y 505.825,Z 709.592,A -85,B 0,C 180,E1 24182.643,E2 24182.643} C_VEL
LIN {X 0,Y 507.006,Z 691.54,A -85,B 0,C 180,E1 24181.722,E2 24181.722} C_VEL
LIN {X 0,Y 508.005,Z 672.092,A -85,B 0,C 180,E1 24180.964,E2 24180.964} C_VEL
LIN {X 0,Y 508.707,Z 652.167,A -85,B 0,C 180,E1 24180.402,E2 24180.402} C_VEL
LIN {X 0,Y 509.238,Z 624.888,A -85,B 0,C 180,E1 24179.92,E2 24179.92} C_VEL
LIN {X 0,Y 512.191,Z 403.731,A -85,B 0,C 180,E1 24176.531,E2 24176.531} C_VEL
LIN {X 0,Y 511.12,Z 399.35,A -85,B 0,C 180,E1 24176.368,E2 24176.368} C_VEL
LIN {X 0,Y 503.685,Z 386.327,A -85,B 0,C 180,E1 24175.468,E2 24175.468} C_VEL
LIN {X 0,Y 497.856,Z 372.026,A -85,B 0,C 180,E1 24173.386,E2 24173.386} C_VEL
LIN {X 0,Y 496.787,Z 369.046,A -85,B 0,C 180,E1 24172.898,E2 24172.898} C_VEL
LIN {X 0,Y 496.738,Z 368.835,A -85,B 0,C 180,E1 24169.363,E2 24169.363} C_VEL
LIN {X 0,Y 496.764,Z 368.85,A -85,B 0,C 180,E1 24165.865,E2 24165.865} C_VEL
LIN {X 0,Y 496.769,Z 368.851,A -85,B 0,C 180,E1 24162.241,E2 24162.241} C_VEL
LIN {X 0,Y 496.732,Z 368.826,A -85,B 0,C 180,E1 24158.839,E2 24158.839} C_VEL
LIN {X 0,Y 496.742,Z 368.858,A -85,B 0,C 180,E1 24155.288,E2 24155.288} C_VEL
LIN {X 0,Y 496.775,Z 368.857,A -85,B 0,C 180,E1 24151.825,E2 24151.825} C_VEL
LIN {X 0,Y 496.734,Z 368.857,A -85,B 0,C 180,E1 24148.362,E2 24148.362} C_VEL
LIN {X 0,Y 496.725,Z 368.857,A -85,B 0,C 180,E1 24144.806,E2 24144.806} C_VEL
LIN {X 0,Y 496.771,Z 368.856,A -85,B 0,C 180,E1 24141.365,E2 24141.365} C_VEL
LIN {X 0,Y 496.744,Z 368.852,A -85,B 0,C 180,E1 24137.828,E2 24137.828} C_VEL
LIN {X 0,Y 496.713,Z 368.854,A -85,B 0,C 180,E1 24134.335,E2 24134.335} C_VEL
LIN {X 0,Y 496.747,Z 368.849,A -85,B 0,C 180,E1 24130.907,E2 24130.907} C_VEL
LIN {X 0,Y 496.737,Z 368.858,A -85,B 0,C 180,E1 24127.518,E2 24127.518} C_VEL
LIN {X 0,Y 496.705,Z 368.86,A -85,B 0,C 180,E1 24124.04,E2 24124.04} C_VEL
LIN {X 0,Y 496.735,Z 368.857,A -85,B 0,C 180,E1 24120.577,E2 24120.577} C_VEL
LIN {X 0,Y 496.725,Z 368.852,A -85,B 0,C 180,E1 24117.231,E2 24117.231} C_VEL
LIN {X 0,Y 496.694,Z 368.857,A -85,B 0,C 180,E1 24113.76,E2 24113.76} C_VEL
LIN {X 0,Y 496.735,Z 368.858,A -85,B 0,C 180,E1 24110.383,E2 24110.383} C_VEL
LIN {X 0,Y 496.716,Z 368.86,A -85,B 0,C 180,E1 24106.949,E2 24106.949} C_VEL
LIN {X 0,Y 496.685,Z 368.862,A -85,B 0,C 180,E1 24103.511,E2 24103.511} C_VEL
LIN {X 0,Y 496.732,Z 368.859,A -85,B 0,C 180,E1 24100.113,E2 24100.113} C_VEL
LIN {X 0,Y 496.697,Z 368.842,A -85,B 0,C 180,E1 24096.888,E2 24096.888} C_VEL
LIN {X 0,Y 496.694,Z 368.863,A -85,B 0,C 180,E1 24093.327,E2 24093.327} C_VEL
LIN {X 0,Y 496.765,Z 368.828,A -85,B 0,C 180,E1 24090.056,E2 24090.056} C_VEL
LIN {X 0,Y 496.706,Z 368.864,A -85,B 0,C 180,E1 24086.648,E2 24086.648} C_VEL
LIN {X 0,Y 496.703,Z 368.852,A -85,B 0,C 180,E1 24083.043,E2 24083.043} C_VEL
LIN {X 0,Y 496.77,Z 368.829,A -85,B 0,C 180,E1 24079.707,E2 24079.707} C_VEL
LIN {X 0,Y 496.722,Z 368.948,A -85,B 0,C 180,E1 24076.496,E2 24076.496} C_VEL
LIN {X 0,Y 497.153,Z 370.615,A -85,B 0,C 180,E1 24076.224,E2 24076.224} C_VEL
LIN {X 0,Y 499.17,Z 374.562,A -85,B 0,C 180,E1 24075.729,E2 24075.729} C_VEL
LIN {X 0,Y 507.718,Z 392.503,A -85,B 0,C 180,E1 24073.638,E2 24073.638} C_VEL
LIN {X 0,Y 514.32,Z 406.782,A -85,B 0,C 180,E1 24072.087,E2 24072.087} C_VEL
LIN {X 0,Y 512.493,Z 453.122,A -85,B 0,C 180,E1 24069.232,E2 24069.232} C_VEL
LIN {X 0,Y 515.418,Z 474.813,A -85,B 0,C 180,E1 24068.625,E2 24068.625} C_VEL
LIN {X 0,Y 512.535,Z 696.23,A -85,B 0,C 180,E1 24065.201,E2 24065.201} C_VEL
LIN {X 0,Y 511.642,Z 762.729,A -85,B 0,C 180,E1 24064.167,E2 24064.167} C_VEL
LIN {X 0,Y 510.835,Z 783.15,A -85,B 0,C 180,E1 24063.656,E2 24063.656} C_VEL
LIN {X 0,Y 509.729,Z 804.793,A -85,B 0,C 180,E1 24062.909,E2 24062.909} C_VEL
LIN {X 0,Y 508.496,Z 825.221,A -85,B 0,C 180,E1 24061.997,E2 24061.997} C_VEL
LIN {X 0,Y 507.026,Z 844.783,A -85,B 0,C 180,E1 24060.908,E2 24060.908} C_VEL
LIN {X 0,Y 505.41,Z 865.529,A -85,B 0,C 180,E1 24059.509,E2 24059.509} C_VEL
LIN {X 0,Y 503.868,Z 883.78,A -85,B 0,C 180,E1 24058.051,E2 24058.051} C_VEL
LIN {X 0,Y 502.31,Z 901.723,A -85,B 0,C 180,E1 24056.35,E2 24056.35} C_VEL
LIN {X 0,Y 500.87,Z 918.179,A -85,B 0,C 180,E1 24054.531,E2 24054.531} C_VEL
LIN {X 0,Y 499.61,Z 933.339,A -85,B 0,C 180,E1 24052.595,E2 24052.595} C_VEL
LIN {X 0,Y 498.487,Z 947.875,A -85,B 0,C 180,E1 24050.425,E2 24050.425} C_VEL
LIN {X 0,Y 497.62,Z 960.192,A -85,B 0,C 180,E1 24048.266,E2 24048.266} C_VEL
LIN {X 0,Y 496.931,Z 971.787,A -85,B 0,C 180,E1 24045.88,E2 24045.88} C_VEL
LIN {X 0,Y 496.469,Z 981.433,A -85,B 0,C 180,E1 24043.509,E2 24043.509} C_VEL
LIN {X 0,Y 496.168,Z 989.416,A -85,B 0,C 180,E1 24041.074,E2 24041.074} C_VEL
LIN {X 0,Y 496.005,Z 996.146,A -85,B 0,C 180,E1 24038.462,E2 24038.462} C_VEL
LIN {X 0,Y 495.937,Z 1000.823,A -85,B 0,C 180,E1 24036.018,E2 24036.018} C_VEL
LIN {X 0,Y 495.913,Z 1003.787,A -85,B 0,C 180,E1 24033.583,E2 24033.583} C_VEL
LIN {X 0,Y 495.908,Z 1005.305,A -85,B 0,C 180,E1 24031.04,E2 24031.04} C_VEL
LIN {X 0,Y 495.908,Z 1005.259,A -85,B 0,C 180,E1 24028.73,E2 24028.73} C_VEL
LIN {X 0,Y 495.911,Z 1003.673,A -85,B 0,C 180,E1 24026.302,E2 24026.302} C_VEL
LIN {X 0,Y 495.941,Z 1000.634,A -85,B 0,C 180,E1 24023.867,E2 24023.867} C_VEL
LIN {X 0,Y 496.009,Z 995.893,A -85,B 0,C 180,E1 24021.422,E2 24021.422} C_VEL
LIN {X 0,Y 496.173,Z 989.179,A -85,B 0,C 180,E1 24018.847,E2 24018.847} C_VEL
LIN {X 0,Y 496.47,Z 981.434,A -85,B 0,C 180,E1 24016.492,E2 24016.492} C_VEL
LIN {X 0,Y 496.936,Z 971.708,A -85,B 0,C 180,E1 24014.102,E2 24014.102} C_VEL
LIN {X 0,Y 497.62,Z 960.197,A -85,B 0,C 180,E1 24011.735,E2 24011.735} C_VEL
LIN {X 0,Y 498.523,Z 947.348,A -85,B 0,C 180,E1 24009.493,E2 24009.493} C_VEL
LIN {X 0,Y 499.609,Z 933.345,A -85,B 0,C 180,E1 24007.406,E2 24007.406} C_VEL
LIN {X 0,Y 500.869,Z 918.187,A -85,B 0,C 180,E1 24005.47,E2 24005.47} C_VEL
LIN {X 0,Y 502.359,Z 901.126,A -85,B 0,C 180,E1 24003.591,E2 24003.591} C_VEL
LIN {X 0,Y 503.93,Z 883.083,A -85,B 0,C 180,E1 24001.889,E2 24001.889} C_VEL
LIN {X 0,Y 505.464,Z 864.912,A -85,B 0,C 180,E1 24000.445,E2 24000.445} C_VEL
LIN {X 0,Y 507.025,Z 844.8,A -85,B 0,C 180,E1 23999.093,E2 23999.093} C_VEL
LIN {X 0,Y 508.495,Z 825.239,A -85,B 0,C 180,E1 23998.004,E2 23998.004} C_VEL
LIN {X 0,Y 509.731,Z 804.792,A -85,B 0,C 180,E1 23997.091,E2 23997.091} C_VEL
LIN {X 0,Y 510.842,Z 783.054,A -85,B 0,C 180,E1 23996.341,E2 23996.341} C_VEL
LIN {X 0,Y 511.648,Z 762.591,A -85,B 0,C 180,E1 23995.83,E2 23995.83} C_VEL
LIN {X 0,Y 512.761,Z 677.874,A -85,B 0,C 180,E1 23994.521,E2 23994.521} C_VEL
LIN {X 0,Y 515.439,Z 473.589,A -85,B 0,C 180,E1 23991.356,E2 23991.356} C_VEL
LIN {X 0,Y 512.427,Z 452.003,A -85,B 0,C 180,E1 23990.721,E2 23990.721} C_VEL
LIN {X 0,Y 514.321,Z 406.783,A -85,B 0,C 180,E1 23987.913,E2 23987.913} C_VEL
LIN {X 0,Y 502.068,Z 380.523,A -85,B 0,C 180,E1 23984.989,E2 23984.989} C_VEL
LIN {X 0,Y 498.053,Z 372.329,A -85,B 0,C 180,E1 23983.995,E2 23983.995} C_VEL
LIN {X 0,Y 496.751,Z 369.126,A -85,B 0,C 180,E1 23983.57,E2 23983.57} C_VEL
LIN {X 0,Y 496.739,Z 368.86,A -85,B 0,C 180,E1 23981.933,E2 23981.933} C_VEL
LIN {X 0,Y 496.728,Z 368.856,A -85,B 0,C 180,E1 23978.608,E2 23978.608} C_VEL
LIN {X 0,Y 496.699,Z 368.84,A -85,B 0,C 180,E1 23975.15,E2 23975.15} C_VEL
LIN {X 0,Y 496.751,Z 368.843,A -85,B 0,C 180,E1 23971.826,E2 23971.826} C_VEL
LIN {X 0,Y 496.7,Z 368.855,A -85,B 0,C 180,E1 23968.626,E2 23968.626} C_VEL
LIN {X 0,Y 496.692,Z 368.837,A -85,B 0,C 180,E1 23965.007,E2 23965.007} C_VEL
LIN {X 0,Y 496.751,Z 368.855,A -85,B 0,C 180,E1 23961.595,E2 23961.595} C_VEL
LIN {X 0,Y 496.699,Z 368.857,A -85,B 0,C 180,E1 23958.18,E2 23958.18} C_VEL
LIN {X 0,Y 496.685,Z 368.859,A -85,B 0,C 180,E1 23954.693,E2 23954.693} C_VEL
LIN {X 0,Y 496.749,Z 368.851,A -85,B 0,C 180,E1 23951.376,E2 23951.376} C_VEL
LIN {X 0,Y 496.696,Z 368.86,A -85,B 0,C 180,E1 23947.984,E2 23947.984} C_VEL
LIN {X 0,Y 496.696,Z 368.86,A -85,B 0,C 180,E1 23944.387,E2 23944.387} C_VEL
LIN {X 0,Y 496.752,Z 368.859,A -85,B 0,C 180,E1 23940.922,E2 23940.922} C_VEL
LIN {X 0,Y 496.713,Z 368.851,A -85,B 0,C 180,E1 23937.577,E2 23937.577} C_VEL
LIN {X 0,Y 496.704,Z 368.848,A -85,B 0,C 180,E1 23934.107,E2 23934.107} C_VEL
LIN {X 0,Y 496.763,Z 368.85,A -85,B 0,C 180,E1 23930.734,E2 23930.734} C_VEL
LIN {X 0,Y 496.72,Z 368.859,A -85,B 0,C 180,E1 23927.325,E2 23927.325} C_VEL
LIN {X 0,Y 496.712,Z 368.858,A -85,B 0,C 180,E1 23923.755,E2 23923.755} C_VEL
LIN {X 0,Y 496.763,Z 368.851,A -85,B 0,C 180,E1 23920.359,E2 23920.359} C_VEL
LIN {X 0,Y 496.729,Z 368.854,A -85,B 0,C 180,E1 23917.014,E2 23917.014} C_VEL
LIN {X 0,Y 496.72,Z 368.853,A -85,B 0,C 180,E1 23913.457,E2 23913.457} C_VEL
LIN {X 0,Y 496.776,Z 368.847,A -85,B 0,C 180,E1 23910.056,E2 23910.056} C_VEL
LIN {X 0,Y 496.75,Z 368.855,A -85,B 0,C 180,E1 23906.529,E2 23906.529} C_VEL
LIN {X 0,Y 496.727,Z 368.856,A -85,B 0,C 180,E1 23902.997,E2 23902.997} C_VEL
LIN {X 0,Y 496.753,Z 368.852,A -85,B 0,C 180,E1 23899.448,E2 23899.448} C_VEL
LIN {X 0,Y 496.768,Z 368.829,A -85,B 0,C 180,E1 23895.928,E2 23895.928} C_VEL
LIN {X 0,Y 496.739,Z 368.847,A -85,B 0,C 180,E1 23892.394,E2 23892.394} C_VEL
LIN {X 0,Y 496.74,Z 368.858,A -85,B 0,C 180,E1 23888.833,E2 23888.833} C_VEL
LIN {X 0,Y 496.766,Z 368.831,A -85,B 0,C 180,E1 23887.452,E2 23887.452} C_VEL
LIN {X 0,Y 496.589,Z 369.571,A -85,B 0,C 180,E1 23887.12,E2 23887.12} C_VEL
LIN {X 0,Y 495.931,Z 372.422,A -85,B 0,C 180,E1 23886.704,E2 23886.704} C_VEL
LIN {X 0,Y 494.385,Z 381.467,A -85,B 0,C 180,E1 23885.86,E2 23885.86} C_VEL
LIN {X 0,Y 494.904,Z 385.117,A -85,B 0,C 180,E1 23885.426,E2 23885.426} C_VEL
LIN {X 0,Y 496.377,Z 388.393,A -85,B 0,C 180,E1 23885.022,E2 23885.022} C_VEL
LIN {X 0,Y 505.486,Z 403.799,A -85,B 0,C 180,E1 23883.949,E2 23883.949} C_VEL
LIN {X 0,Y 505.781,Z 407.837,A -85,B 0,C 180,E1 23883.856,E2 23883.856} C_VEL
LIN {X 0,Y 502.453,Z 640.004,A -85,B 0,C 180,E1 23880.276,E2 23880.276} C_VEL
LIN {X 0,Y 501.95,Z 660.447,A -85,B 0,C 180,E1 23879.834,E2 23879.834} C_VEL
LIN {X 0,Y 501.014,Z 680.644,A -85,B 0,C 180,E1 23879.177,E2 23879.177} C_VEL
LIN {X 0,Y 499.912,Z 699.329,A -85,B 0,C 180,E1 23878.353,E2 23878.353} C_VEL
LIN {X 0,Y 498.48,Z 718.569,A -85,B 0,C 180,E1 23877.276,E2 23877.276} C_VEL
LIN {X 0,Y 497.004,Z 735.918,A -85,B 0,C 180,E1 23876.073,E2 23876.073} C_VEL
LIN {X 0,Y 495.442,Z 752.489,A -85,B 0,C 180,E1 23874.689,E2 23874.689} C_VEL
LIN {X 0,Y 493.81,Z 768.659,A -85,B 0,C 180,E1 23873.063,E2 23873.063} C_VEL
LIN {X 0,Y 492.313,Z 783.259,A -85,B 0,C 180,E1 23871.315,E2 23871.315} C_VEL
LIN {X 0,Y 490.936,Z 796.875,A -85,B 0,C 180,E1 23869.386,E2 23869.386} C_VEL
LIN {X 0,Y 489.757,Z 809.996,A -85,B 0,C 180,E1 23867.168,E2 23867.168} C_VEL
LIN {X 0,Y 489.007,Z 821.708,A -85,B 0,C 180,E1 23864.927,E2 23864.927} C_VEL
LIN {X 0,Y 488.506,Z 831.596,A -85,B 0,C 180,E1 23862.649,E2 23862.649} C_VEL
LIN {X 0,Y 488.187,Z 839.585,A -85,B 0,C 180,E1 23860.382,E2 23860.382} C_VEL
LIN {X 0,Y 488.019,Z 846.102,A -85,B 0,C 180,E1 23858.007,E2 23858.007} C_VEL
LIN {X 0,Y 487.935,Z 850.8,A -85,B 0,C 180,E1 23855.644,E2 23855.644} C_VEL
LIN {X 0,Y 487.903,Z 853.85,A -85,B 0,C 180,E1 23853.289,E2 23853.289} C_VEL
LIN {X 0,Y 487.911,Z 855.318,A -85,B 0,C 180,E1 23850.939,E2 23850.939} C_VEL
LIN {X 0,Y 487.901,Z 855.233,A -85,B 0,C 180,E1 23848.591,E2 23848.591} C_VEL
LIN {X 0,Y 487.912,Z 853.48,A -85,B 0,C 180,E1 23846.24,E2 23846.24} C_VEL
LIN {X 0,Y 487.951,Z 850.131,A -85,B 0,C 180,E1 23843.884,E2 23843.884} C_VEL
LIN {X 0,Y 488.041,Z 845.125,A -85,B 0,C 180,E1 23841.518,E2 23841.518} C_VEL
LIN {X 0,Y 488.224,Z 838.744,A -85,B 0,C 180,E1 23839.26,E2 23839.26} C_VEL
LIN {X 0,Y 488.584,Z 830.095,A -85,B 0,C 180,E1 23836.871,E2 23836.871} C_VEL
LIN {X 0,Y 489.121,Z 819.83,A -85,B 0,C 180,E1 23834.59,E2 23834.59} C_VEL
LIN {X 0,Y 490.198,Z 804.819,A -85,B 0,C 180,E1 23831.817,E2 23831.817} C_VEL
LIN {X 0,Y 491.374,Z 792.701,A -85,B 0,C 180,E1 23829.888,E2 23829.888} C_VEL
LIN {X 0,Y 492.877,Z 777.777,A -85,B 0,C 180,E1 23827.897,E2 23827.897} C_VEL
LIN {X 0,Y 494.481,Z 762.054,A -85,B 0,C 180,E1 23826.148,E2 23826.148} C_VEL
LIN {X 0,Y 496.065,Z 745.866,A -85,B 0,C 180,E1 23824.642,E2 23824.642} C_VEL
LIN {X 0,Y 497.618,Z 728.829,A -85,B 0,C 180,E1 23823.318,E2 23823.318} C_VEL
LIN {X 0,Y 499.084,Z 710.967,A -85,B 0,C 180,E1 23822.177,E2 23822.177} C_VEL
LIN {X 0,Y 500.337,Z 692.937,A -85,B 0,C 180,E1 23821.245,E2 23821.245} C_VEL
LIN {X 0,Y 501.387,Z 673.507,A -85,B 0,C 180,E1 23820.477,E2 23820.477} C_VEL
LIN {X 0,Y 502.127,Z 653.524,A -85,B 0,C 180,E1 23819.905,E2 23819.905} C_VEL
LIN {X 0,Y 502.66,Z 627.269,A -85,B 0,C 180,E1 23819.432,E2 23819.432} C_VEL
LIN {X 0,Y 505.803,Z 405.415,A -85,B 0,C 180,E1 23816.015,E2 23816.015} C_VEL
LIN {X 0,Y 505.026,Z 402.92,A -85,B 0,C 180,E1 23815.905,E2 23815.905} C_VEL
LIN {X 0,Y 495.793,Z 387.189,A -85,B 0,C 180,E1 23814.78,E2 23814.78} C_VEL
LIN {X 0,Y 489.694,Z 372.572,A -85,B 0,C 180,E1 23812.586,E2 23812.586} C_VEL
LIN {X 0,Y 488.851,Z 369.985,A -85,B 0,C 180,E1 23812.139,E2 23812.139} C_VEL
LIN {X 0,Y 488.831,Z 369.816,A -85,B 0,C 180,E1 23808.471,E2 23808.471} C_VEL
LIN {X 0,Y 488.8,Z 369.825,A -85,B 0,C 180,E1 23804.953,E2 23804.953} C_VEL
LIN {X 0,Y 488.803,Z 369.848,A -85,B 0,C 180,E1 23801.354,E2 23801.354} C_VEL
LIN {X 0,Y 488.829,Z 369.815,A -85,B 0,C 180,E1 23797.852,E2 23797.852} C_VEL
LIN {X 0,Y 488.815,Z 369.84,A -85,B 0,C 180,E1 23794.28,E2 23794.28} C_VEL
LIN {X 0,Y 488.787,Z 369.838,A -85,B 0,C 180,E1 23790.757,E2 23790.757} C_VEL
LIN {X 0,Y 488.812,Z 369.838,A -85,B 0,C 180,E1 23787.271,E2 23787.271} C_VEL
LIN {X 0,Y 488.826,Z 369.84,A -85,B 0,C 180,E1 23783.763,E2 23783.763} C_VEL
LIN {X 0,Y 488.781,Z 369.844,A -85,B 0,C 180,E1 23780.35,E2 23780.35} C_VEL
